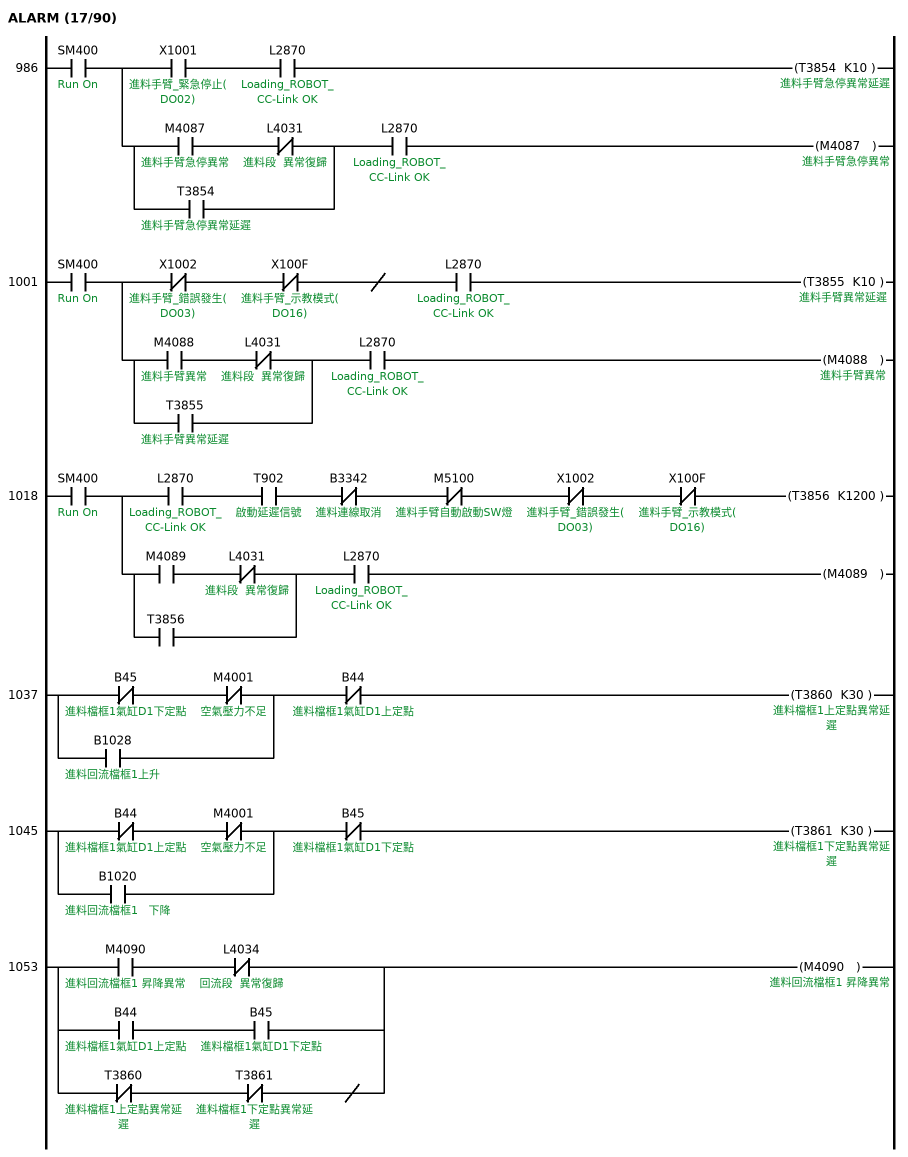
[picture p192: ladder of ALARM, rungs at steps 986 to 1053]
986   LD      SM400  ; Run On
      MPS
      AND     X1001  ; 進料手臂_緊急停止(DO02)
      AND     L2870  ; Loading_ROBOT_  CC-Link OK
      OUT     T3854 K10  ; 進料手臂急停異常延遲
      MPP
      LD      M4087  ; 進料手臂急停異常
      ANI     L4031  ; 進料段  異常復歸
      OR      T3854  ; 進料手臂急停異常延遲
      ANB
      AND     L2870  ; Loading_ROBOT_  CC-Link OK
      OUT     M4087  ; 進料手臂急停異常
1001  LD      SM400  ; Run On
      MPS
      ANI     X1002  ; 進料手臂_錯誤發生(DO03)
      ANI     X100F  ; 進料手臂_示教模式(DO16)
      INV
      AND     L2870  ; Loading_ROBOT_  CC-Link OK
      OUT     T3855 K10  ; 進料手臂異常延遲
      MPP
      LD      M4088  ; 進料手臂異常
      ANI     L4031  ; 進料段  異常復歸
      OR      T3855  ; 進料手臂異常延遲
      ANB
      AND     L2870  ; Loading_ROBOT_  CC-Link OK
      OUT     M4088  ; 進料手臂異常
1018  LD      SM400  ; Run On
      MPS
      AND     L2870  ; Loading_ROBOT_  CC-Link OK
      AND     T902  ; 啟動延遲信號
      ANI     B3342  ; 進料連線取消
      ANI     M5100  ; 進料手臂自動啟動SW燈
      ANI     X1002  ; 進料手臂_錯誤發生(DO03)
      ANI     X100F  ; 進料手臂_示教模式(DO16)
      OUT     T3856 K1200
      MPP
      LD      M4089
      ANI     L4031  ; 進料段  異常復歸
      OR      T3856
      ANB
      AND     L2870  ; Loading_ROBOT_  CC-Link OK
      OUT     M4089
1037  LDI     B45  ; 進料檔框1氣缸D1下定點
      ANI     M4001  ; 空氣壓力不足
      OR      B1028  ; 進料回流檔框1上升
      ANI     B44  ; 進料檔框1氣缸D1上定點
      OUT     T3860 K30  ; 進料檔框1上定點異常延遲
1045  LDI     B44  ; 進料檔框1氣缸D1上定點
      ANI     M4001  ; 空氣壓力不足
      OR      B1020  ; 進料回流檔框1   下降
      ANI     B45  ; 進料檔框1氣缸D1下定點
      OUT     T3861 K30  ; 進料檔框1下定點異常延遲
1053  LD      M4090  ; 進料回流檔框1 昇降異常
      ANI     L4034  ; 回流段  異常復歸
      LD      B44  ; 進料檔框1氣缸D1上定點
      AND     B45  ; 進料檔框1氣缸D1下定點
      ORB
      LDI     T3860  ; 進料檔框1上定點異常延遲
      ANI     T3861  ; 進料檔框1下定點異常延遲
      INV
      ORB
      OUT     M4090  ; 進料回流檔框1 昇降異常
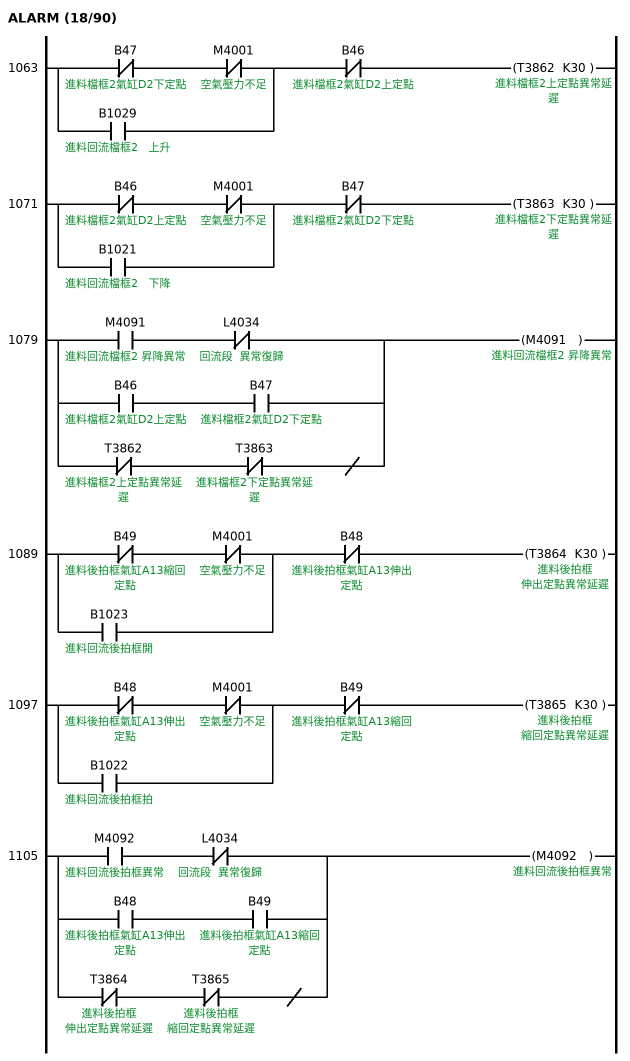
1063  LDI     B47  ; 進料檔框2氣缸D2下定點
      ANI     M4001  ; 空氣壓力不足
      OR      B1029  ; 進料回流檔框2   上升
      ANI     B46  ; 進料檔框2氣缸D2上定點
      OUT     T3862 K30  ; 進料檔框2上定點異常延遲
1071  LDI     B46  ; 進料檔框2氣缸D2上定點
      ANI     M4001  ; 空氣壓力不足
      OR      B1021  ; 進料回流檔框2   下降
      ANI     B47  ; 進料檔框2氣缸D2下定點
      OUT     T3863 K30  ; 進料檔框2下定點異常延遲
1079  LD      M4091  ; 進料回流檔框2 昇降異常
      ANI     L4034  ; 回流段  異常復歸
      LD      B46  ; 進料檔框2氣缸D2上定點
      AND     B47  ; 進料檔框2氣缸D2下定點
      ORB
      LDI     T3862  ; 進料檔框2上定點異常延遲
      ANI     T3863  ; 進料檔框2下定點異常延遲
      INV
      ORB
      OUT     M4091  ; 進料回流檔框2 昇降異常
1089  LDI     B49  ; 進料後拍框氣缸A13縮回定點
      ANI     M4001  ; 空氣壓力不足
      OR      B1023  ; 進料回流後拍框開
      ANI     B48  ; 進料後拍框氣缸A13伸出定點
      OUT     T3864 K30  ; 進料後拍框    伸出定點異常延遲
1097  LDI     B48  ; 進料後拍框氣缸A13伸出定點
      ANI     M4001  ; 空氣壓力不足
      OR      B1022  ; 進料回流後拍框拍
      ANI     B49  ; 進料後拍框氣缸A13縮回定點
      OUT     T3865 K30  ; 進料後拍框    縮回定點異常延遲
1105  LD      M4092  ; 進料回流後拍框異常
      ANI     L4034  ; 回流段  異常復歸
      LD      B48  ; 進料後拍框氣缸A13伸出定點
      AND     B49  ; 進料後拍框氣缸A13縮回定點
      ORB
      LDI     T3864  ; 進料後拍框    伸出定點異常延遲
      ANI     T3865  ; 進料後拍框    縮回定點異常延遲
      INV
      ORB
      OUT     M4092  ; 進料回流後拍框異常
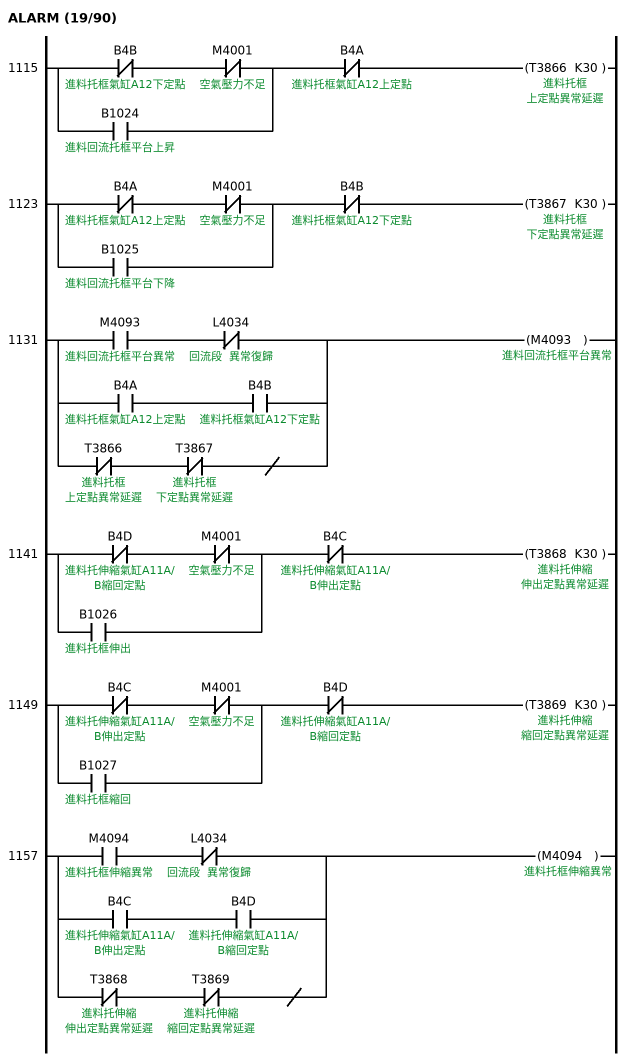
1115  LDI     B4B  ; 進料托框氣缸A12下定點
      ANI     M4001  ; 空氣壓力不足
      OR      B1024  ; 進料回流托框平台上昇
      ANI     B4A  ; 進料托框氣缸A12上定點
      OUT     T3866 K30  ; 進料托框    上定點異常延遲
1123  LDI     B4A  ; 進料托框氣缸A12上定點
      ANI     M4001  ; 空氣壓力不足
      OR      B1025  ; 進料回流托框平台下降
      ANI     B4B  ; 進料托框氣缸A12下定點
      OUT     T3867 K30  ; 進料托框    下定點異常延遲
1131  LD      M4093  ; 進料回流托框平台異常
      ANI     L4034  ; 回流段  異常復歸
      LD      B4A  ; 進料托框氣缸A12上定點
      AND     B4B  ; 進料托框氣缸A12下定點
      ORB
      LDI     T3866  ; 進料托框    上定點異常延遲
      ANI     T3867  ; 進料托框    下定點異常延遲
      INV
      ORB
      OUT     M4093  ; 進料回流托框平台異常
1141  LDI     B4D  ; 進料托伸縮氣缸A11A/B縮回定點
      ANI     M4001  ; 空氣壓力不足
      OR      B1026  ; 進料托框伸出
      ANI     B4C  ; 進料托伸縮氣缸A11A/B伸出定點
      OUT     T3868 K30  ; 進料托伸縮    伸出定點異常延遲
1149  LDI     B4C  ; 進料托伸縮氣缸A11A/B伸出定點
      ANI     M4001  ; 空氣壓力不足
      OR      B1027  ; 進料托框縮回
      ANI     B4D  ; 進料托伸縮氣缸A11A/B縮回定點
      OUT     T3869 K30  ; 進料托伸縮    縮回定點異常延遲
1157  LD      M4094  ; 進料托框伸縮異常
      ANI     L4034  ; 回流段  異常復歸
      LD      B4C  ; 進料托伸縮氣缸A11A/B伸出定點
      AND     B4D  ; 進料托伸縮氣缸A11A/B縮回定點
      ORB
      LDI     T3868  ; 進料托伸縮    伸出定點異常延遲
      ANI     T3869  ; 進料托伸縮    縮回定點異常延遲
      INV
      ORB
      OUT     M4094  ; 進料托框伸縮異常
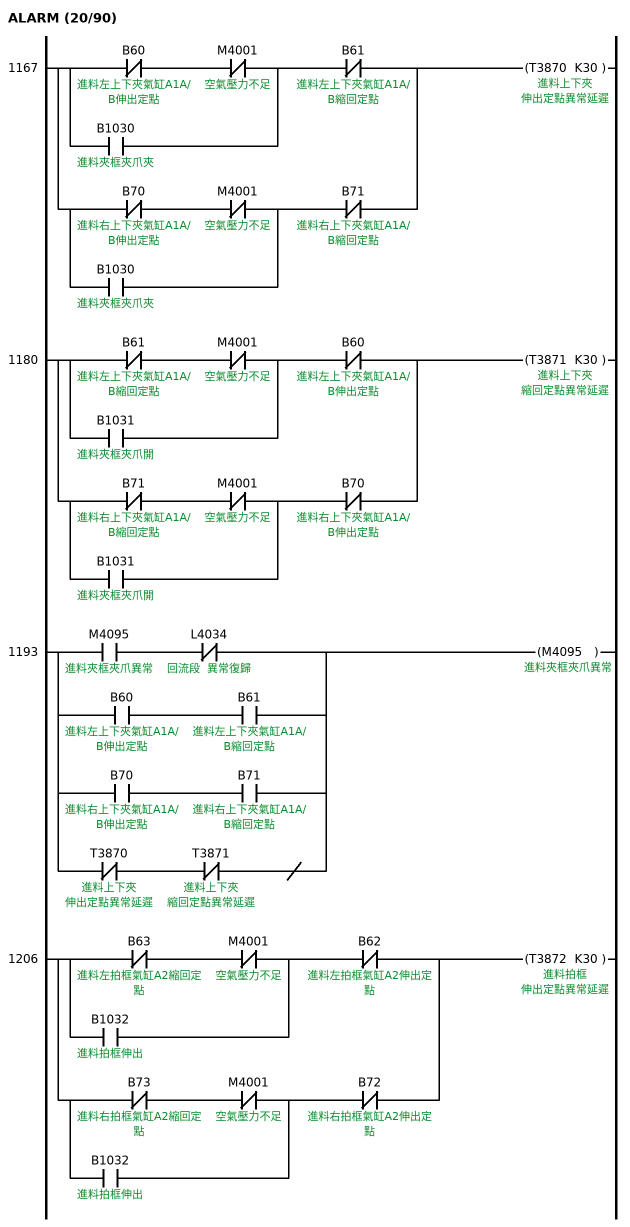
1167  LDI     B60  ; 進料左上下夾氣缸A1A/B伸出定點
      ANI     M4001  ; 空氣壓力不足
      OR      B1030  ; 進料夾框夾爪夾
      ANI     B61  ; 進料左上下夾氣缸A1A/B縮回定點
      LDI     B70  ; 進料右上下夾氣缸A1A/B伸出定點
      ANI     M4001  ; 空氣壓力不足
      OR      B1030  ; 進料夾框夾爪夾
      ANI     B71  ; 進料右上下夾氣缸A1A/B縮回定點
      ORB
      OUT     T3870 K30  ; 進料上下夾    伸出定點異常延遲
1180  LDI     B61  ; 進料左上下夾氣缸A1A/B縮回定點
      ANI     M4001  ; 空氣壓力不足
      OR      B1031  ; 進料夾框夾爪開
      ANI     B60  ; 進料左上下夾氣缸A1A/B伸出定點
      LDI     B71  ; 進料右上下夾氣缸A1A/B縮回定點
      ANI     M4001  ; 空氣壓力不足
      OR      B1031  ; 進料夾框夾爪開
      ANI     B70  ; 進料右上下夾氣缸A1A/B伸出定點
      ORB
      OUT     T3871 K30  ; 進料上下夾    縮回定點異常延遲
1193  LD      M4095  ; 進料夾框夾爪異常
      ANI     L4034  ; 回流段  異常復歸
      LD      B60  ; 進料左上下夾氣缸A1A/B伸出定點
      AND     B61  ; 進料左上下夾氣缸A1A/B縮回定點
      ORB
      LD      B70  ; 進料右上下夾氣缸A1A/B伸出定點
      AND     B71  ; 進料右上下夾氣缸A1A/B縮回定點
      ORB
      LDI     T3870  ; 進料上下夾    伸出定點異常延遲
      ANI     T3871  ; 進料上下夾    縮回定點異常延遲
      INV
      ORB
      OUT     M4095  ; 進料夾框夾爪異常
1206  LDI     B63  ; 進料左拍框氣缸A2縮回定點
      ANI     M4001  ; 空氣壓力不足
      OR      B1032  ; 進料拍框伸出
      ANI     B62  ; 進料左拍框氣缸A2伸出定點
      LDI     B73  ; 進料右拍框氣缸A2縮回定點
      ANI     M4001  ; 空氣壓力不足
      OR      B1032  ; 進料拍框伸出
      ANI     B72  ; 進料右拍框氣缸A2伸出定點
      ORB
      OUT     T3872 K30  ; 進料拍框    伸出定點異常延遲
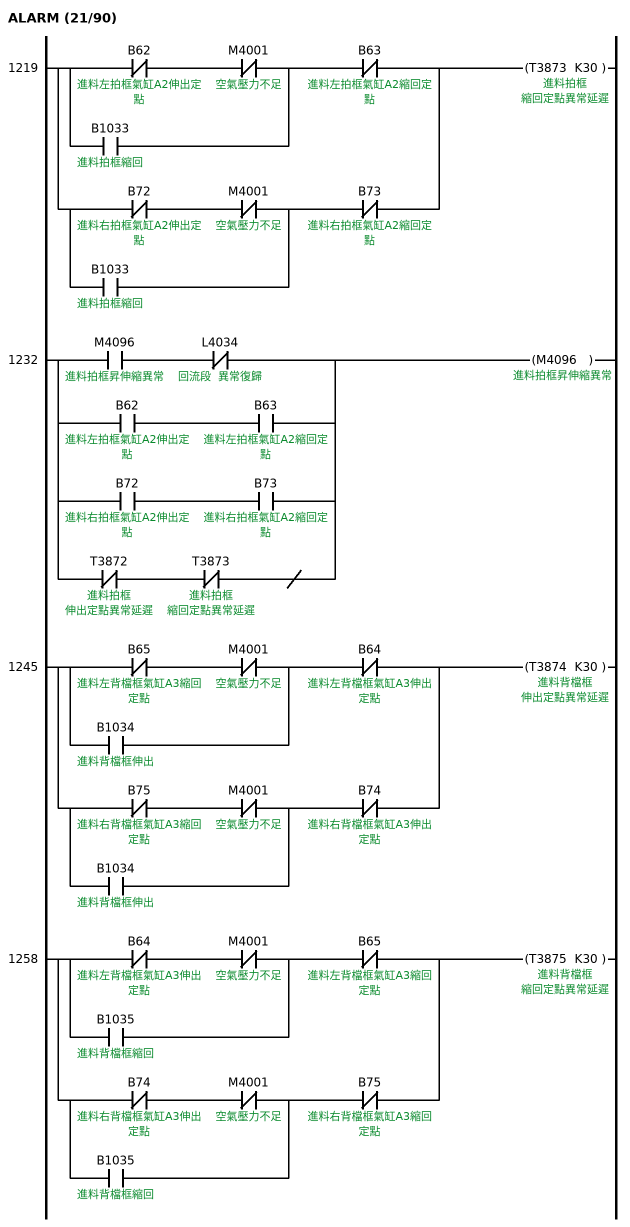
1219  LDI     B62  ; 進料左拍框氣缸A2伸出定點
      ANI     M4001  ; 空氣壓力不足
      OR      B1033  ; 進料拍框縮回
      ANI     B63  ; 進料左拍框氣缸A2縮回定點
      LDI     B72  ; 進料右拍框氣缸A2伸出定點
      ANI     M4001  ; 空氣壓力不足
      OR      B1033  ; 進料拍框縮回
      ANI     B73  ; 進料右拍框氣缸A2縮回定點
      ORB
      OUT     T3873 K30  ; 進料拍框    縮回定點異常延遲
1232  LD      M4096  ; 進料拍框昇伸縮異常
      ANI     L4034  ; 回流段  異常復歸
      LD      B62  ; 進料左拍框氣缸A2伸出定點
      AND     B63  ; 進料左拍框氣缸A2縮回定點
      ORB
      LD      B72  ; 進料右拍框氣缸A2伸出定點
      AND     B73  ; 進料右拍框氣缸A2縮回定點
      ORB
      LDI     T3872  ; 進料拍框    伸出定點異常延遲
      ANI     T3873  ; 進料拍框    縮回定點異常延遲
      INV
      ORB
      OUT     M4096  ; 進料拍框昇伸縮異常
1245  LDI     B65  ; 進料左背檔框氣缸A3縮回定點
      ANI     M4001  ; 空氣壓力不足
      OR      B1034  ; 進料背檔框伸出
      ANI     B64  ; 進料左背檔框氣缸A3伸出定點
      LDI     B75  ; 進料右背檔框氣缸A3縮回定點
      ANI     M4001  ; 空氣壓力不足
      OR      B1034  ; 進料背檔框伸出
      ANI     B74  ; 進料右背檔框氣缸A3伸出定點
      ORB
      OUT     T3874 K30  ; 進料背檔框    伸出定點異常延遲
1258  LDI     B64  ; 進料左背檔框氣缸A3伸出定點
      ANI     M4001  ; 空氣壓力不足
      OR      B1035  ; 進料背檔框縮回
      ANI     B65  ; 進料左背檔框氣缸A3縮回定點
      LDI     B74  ; 進料右背檔框氣缸A3伸出定點
      ANI     M4001  ; 空氣壓力不足
      OR      B1035  ; 進料背檔框縮回
      ANI     B75  ; 進料右背檔框氣缸A3縮回定點
      ORB
      OUT     T3875 K30  ; 進料背檔框    縮回定點異常延遲
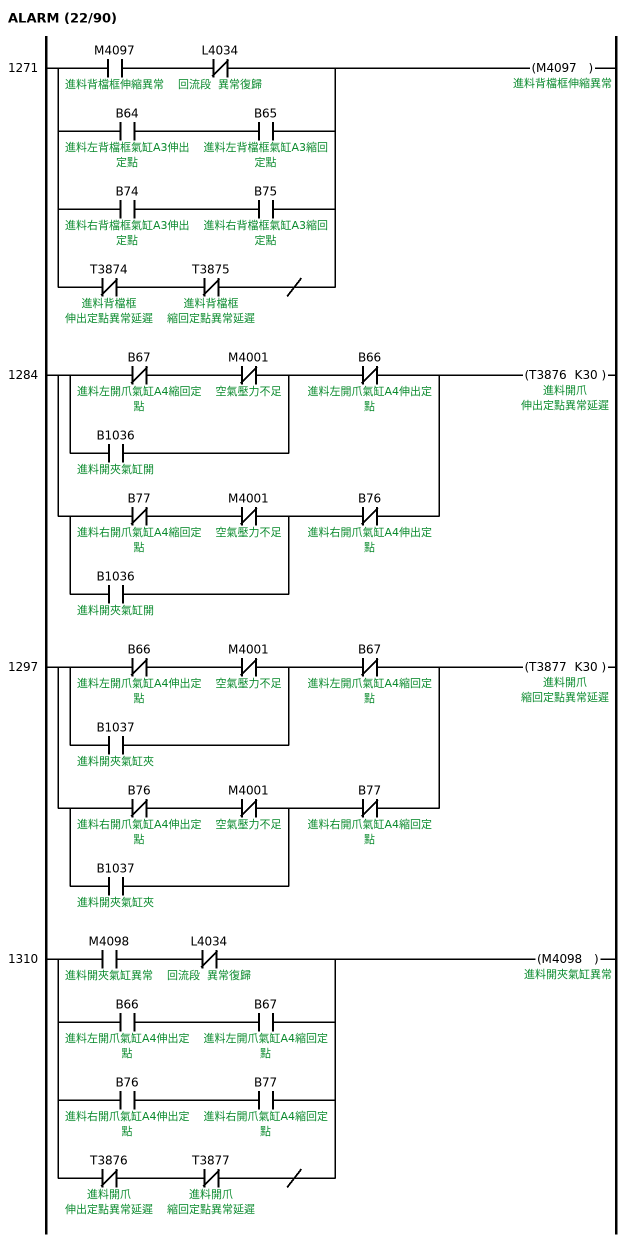
1271  LD      M4097  ; 進料背檔框伸縮異常
      ANI     L4034  ; 回流段  異常復歸
      LD      B64  ; 進料左背檔框氣缸A3伸出定點
      AND     B65  ; 進料左背檔框氣缸A3縮回定點
      ORB
      LD      B74  ; 進料右背檔框氣缸A3伸出定點
      AND     B75  ; 進料右背檔框氣缸A3縮回定點
      ORB
      LDI     T3874  ; 進料背檔框    伸出定點異常延遲
      ANI     T3875  ; 進料背檔框    縮回定點異常延遲
      INV
      ORB
      OUT     M4097  ; 進料背檔框伸縮異常
1284  LDI     B67  ; 進料左開爪氣缸A4縮回定點
      ANI     M4001  ; 空氣壓力不足
      OR      B1036  ; 進料開夾氣缸開
      ANI     B66  ; 進料左開爪氣缸A4伸出定點
      LDI     B77  ; 進料右開爪氣缸A4縮回定點
      ANI     M4001  ; 空氣壓力不足
      OR      B1036  ; 進料開夾氣缸開
      ANI     B76  ; 進料右開爪氣缸A4伸出定點
      ORB
      OUT     T3876 K30  ; 進料開爪    伸出定點異常延遲
1297  LDI     B66  ; 進料左開爪氣缸A4伸出定點
      ANI     M4001  ; 空氣壓力不足
      OR      B1037  ; 進料開夾氣缸夾
      ANI     B67  ; 進料左開爪氣缸A4縮回定點
      LDI     B76  ; 進料右開爪氣缸A4伸出定點
      ANI     M4001  ; 空氣壓力不足
      OR      B1037  ; 進料開夾氣缸夾
      ANI     B77  ; 進料右開爪氣缸A4縮回定點
      ORB
      OUT     T3877 K30  ; 進料開爪    縮回定點異常延遲
1310  LD      M4098  ; 進料開夾氣缸異常
      ANI     L4034  ; 回流段  異常復歸
      LD      B66  ; 進料左開爪氣缸A4伸出定點
      AND     B67  ; 進料左開爪氣缸A4縮回定點
      ORB
      LD      B76  ; 進料右開爪氣缸A4伸出定點
      AND     B77  ; 進料右開爪氣缸A4縮回定點
      ORB
      LDI     T3876  ; 進料開爪    伸出定點異常延遲
      ANI     T3877  ; 進料開爪    縮回定點異常延遲
      INV
      ORB
      OUT     M4098  ; 進料開夾氣缸異常
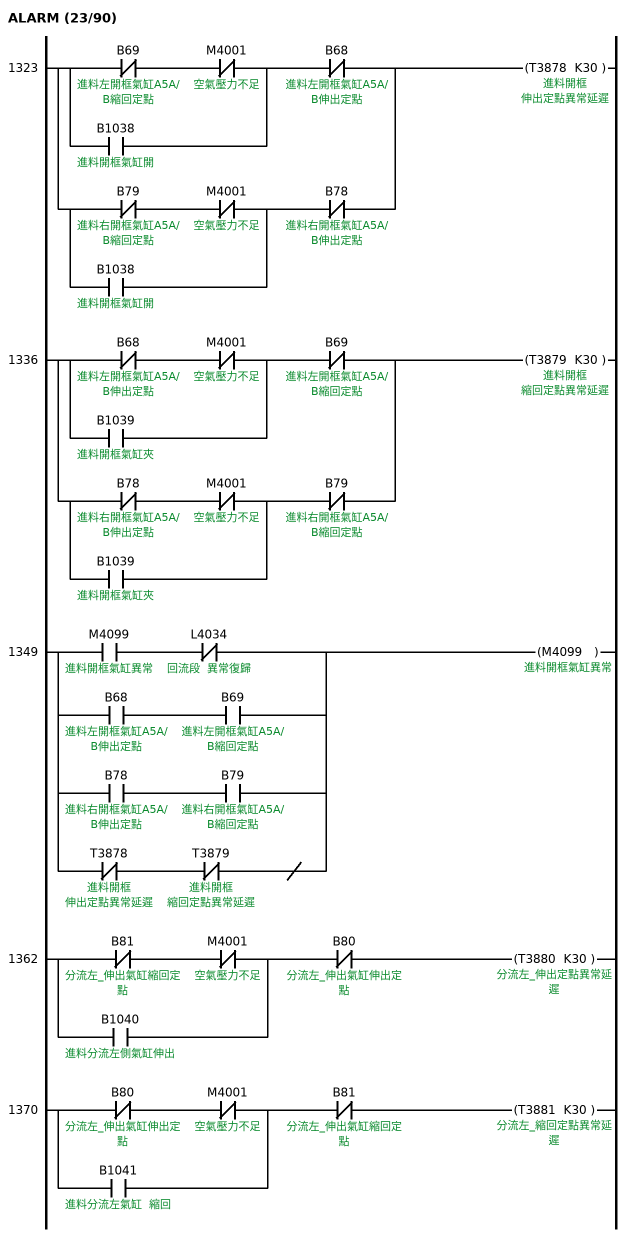
1323  LDI     B69  ; 進料左開框氣缸A5A/B縮回定點
      ANI     M4001  ; 空氣壓力不足
      OR      B1038  ; 進料開框氣缸開
      ANI     B68  ; 進料左開框氣缸A5A/B伸出定點
      LDI     B79  ; 進料右開框氣缸A5A/B縮回定點
      ANI     M4001  ; 空氣壓力不足
      OR      B1038  ; 進料開框氣缸開
      ANI     B78  ; 進料右開框氣缸A5A/B伸出定點
      ORB
      OUT     T3878 K30  ; 進料開框    伸出定點異常延遲
1336  LDI     B68  ; 進料左開框氣缸A5A/B伸出定點
      ANI     M4001  ; 空氣壓力不足
      OR      B1039  ; 進料開框氣缸夾
      ANI     B69  ; 進料左開框氣缸A5A/B縮回定點
      LDI     B78  ; 進料右開框氣缸A5A/B伸出定點
      ANI     M4001  ; 空氣壓力不足
      OR      B1039  ; 進料開框氣缸夾
      ANI     B79  ; 進料右開框氣缸A5A/B縮回定點
      ORB
      OUT     T3879 K30  ; 進料開框    縮回定點異常延遲
1349  LD      M4099  ; 進料開框氣缸異常
      ANI     L4034  ; 回流段  異常復歸
      LD      B68  ; 進料左開框氣缸A5A/B伸出定點
      AND     B69  ; 進料左開框氣缸A5A/B縮回定點
      ORB
      LD      B78  ; 進料右開框氣缸A5A/B伸出定點
      AND     B79  ; 進料右開框氣缸A5A/B縮回定點
      ORB
      LDI     T3878  ; 進料開框    伸出定點異常延遲
      ANI     T3879  ; 進料開框    縮回定點異常延遲
      INV
      ORB
      OUT     M4099  ; 進料開框氣缸異常
1362  LDI     B81  ; 分流左_伸出氣缸縮回定點
      ANI     M4001  ; 空氣壓力不足
      OR      B1040  ; 進料分流左側氣缸伸出
      ANI     B80  ; 分流左_伸出氣缸伸出定點
      OUT     T3880 K30  ; 分流左_伸出定點異常延遲
1370  LDI     B80  ; 分流左_伸出氣缸伸出定點
      ANI     M4001  ; 空氣壓力不足
      OR      B1041  ; 進料分流左氣缸  縮回
      ANI     B81  ; 分流左_伸出氣缸縮回定點
      OUT     T3881 K30  ; 分流左_縮回定點異常延遲
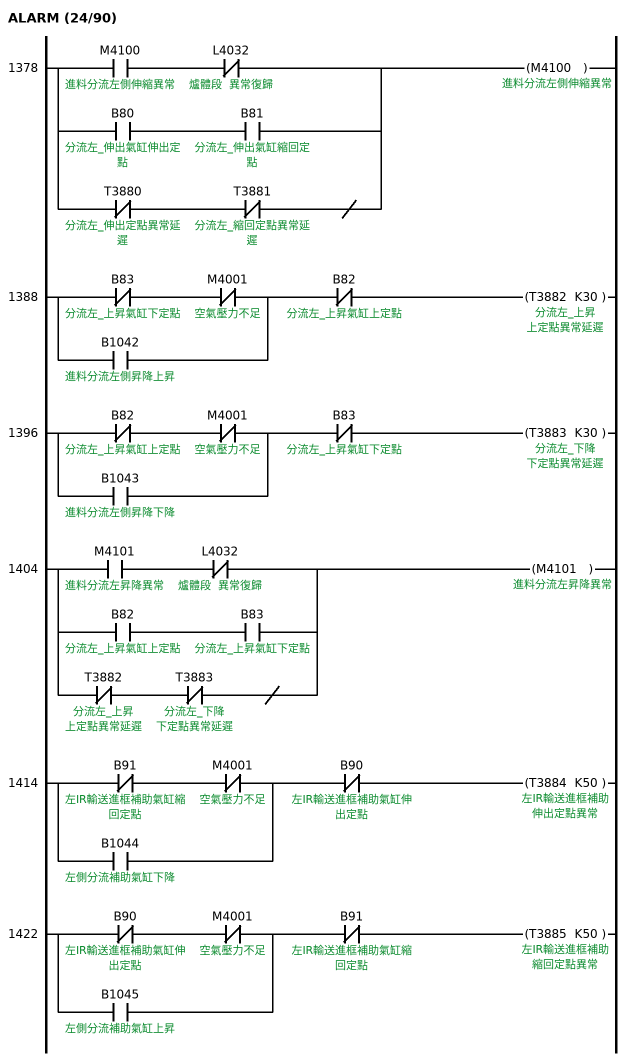
1378  LD      M4100  ; 進料分流左側伸縮異常
      ANI     L4032  ; 爐體段  異常復歸
      LD      B80  ; 分流左_伸出氣缸伸出定點
      AND     B81  ; 分流左_伸出氣缸縮回定點
      ORB
      LDI     T3880  ; 分流左_伸出定點異常延遲
      ANI     T3881  ; 分流左_縮回定點異常延遲
      INV
      ORB
      OUT     M4100  ; 進料分流左側伸縮異常
1388  LDI     B83  ; 分流左_上昇氣缸下定點
      ANI     M4001  ; 空氣壓力不足
      OR      B1042  ; 進料分流左側昇降上昇
      ANI     B82  ; 分流左_上昇氣缸上定點
      OUT     T3882 K30  ; 分流左_上昇    上定點異常延遲
1396  LDI     B82  ; 分流左_上昇氣缸上定點
      ANI     M4001  ; 空氣壓力不足
      OR      B1043  ; 進料分流左側昇降下降
      ANI     B83  ; 分流左_上昇氣缸下定點
      OUT     T3883 K30  ; 分流左_下降    下定點異常延遲
1404  LD      M4101  ; 進料分流左昇降異常
      ANI     L4032  ; 爐體段  異常復歸
      LD      B82  ; 分流左_上昇氣缸上定點
      AND     B83  ; 分流左_上昇氣缸下定點
      ORB
      LDI     T3882  ; 分流左_上昇    上定點異常延遲
      ANI     T3883  ; 分流左_下降    下定點異常延遲
      INV
      ORB
      OUT     M4101  ; 進料分流左昇降異常
1414  LDI     B91  ; 左IR輸送進框補助氣缸縮回定點
      ANI     M4001  ; 空氣壓力不足
      OR      B1044  ; 左側分流補助氣缸下降
      ANI     B90  ; 左IR輸送進框補助氣缸伸出定點
      OUT     T3884 K50  ; 左IR輸送進框補助    伸出定點異常
1422  LDI     B90  ; 左IR輸送進框補助氣缸伸出定點
      ANI     M4001  ; 空氣壓力不足
      OR      B1045  ; 左側分流補助氣缸上昇
      ANI     B91  ; 左IR輸送進框補助氣缸縮回定點
      OUT     T3885 K50  ; 左IR輸送進框補助    縮回定點異常
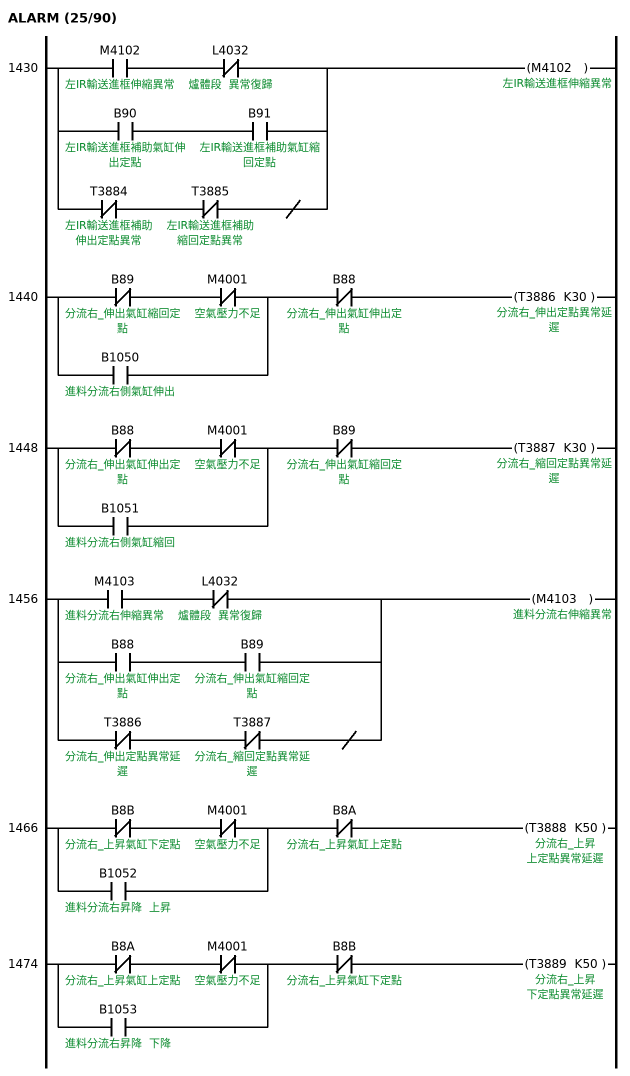
1430  LD      M4102  ; 左IR輸送進框伸縮異常
      ANI     L4032  ; 爐體段  異常復歸
      LD      B90  ; 左IR輸送進框補助氣缸伸出定點
      AND     B91  ; 左IR輸送進框補助氣缸縮回定點
      ORB
      LDI     T3884  ; 左IR輸送進框補助    伸出定點異常
      ANI     T3885  ; 左IR輸送進框補助    縮回定點異常
      INV
      ORB
      OUT     M4102  ; 左IR輸送進框伸縮異常
1440  LDI     B89  ; 分流右_伸出氣缸縮回定點
      ANI     M4001  ; 空氣壓力不足
      OR      B1050  ; 進料分流右側氣缸伸出
      ANI     B88  ; 分流右_伸出氣缸伸出定點
      OUT     T3886 K30  ; 分流右_伸出定點異常延遲
1448  LDI     B88  ; 分流右_伸出氣缸伸出定點
      ANI     M4001  ; 空氣壓力不足
      OR      B1051  ; 進料分流右側氣缸縮回
      ANI     B89  ; 分流右_伸出氣缸縮回定點
      OUT     T3887 K30  ; 分流右_縮回定點異常延遲
1456  LD      M4103  ; 進料分流右伸縮異常
      ANI     L4032  ; 爐體段  異常復歸
      LD      B88  ; 分流右_伸出氣缸伸出定點
      AND     B89  ; 分流右_伸出氣缸縮回定點
      ORB
      LDI     T3886  ; 分流右_伸出定點異常延遲
      ANI     T3887  ; 分流右_縮回定點異常延遲
      INV
      ORB
      OUT     M4103  ; 進料分流右伸縮異常
1466  LDI     B8B  ; 分流右_上昇氣缸下定點
      ANI     M4001  ; 空氣壓力不足
      OR      B1052  ; 進料分流右昇降  上昇
      ANI     B8A  ; 分流右_上昇氣缸上定點
      OUT     T3888 K50  ; 分流右_上昇    上定點異常延遲
1474  LDI     B8A  ; 分流右_上昇氣缸上定點
      ANI     M4001  ; 空氣壓力不足
      OR      B1053  ; 進料分流右昇降  下降
      ANI     B8B  ; 分流右_上昇氣缸下定點
      OUT     T3889 K50  ; 分流右_上昇    下定點異常延遲
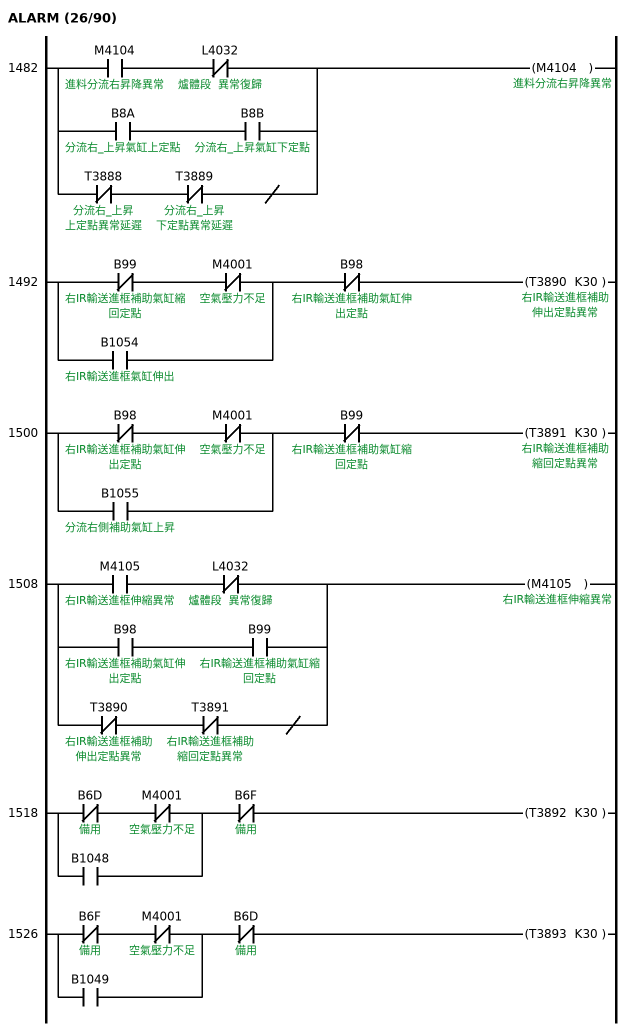
1482  LD      M4104  ; 進料分流右昇降異常
      ANI     L4032  ; 爐體段  異常復歸
      LD      B8A  ; 分流右_上昇氣缸上定點
      AND     B8B  ; 分流右_上昇氣缸下定點
      ORB
      LDI     T3888  ; 分流右_上昇    上定點異常延遲
      ANI     T3889  ; 分流右_上昇    下定點異常延遲
      INV
      ORB
      OUT     M4104  ; 進料分流右昇降異常
1492  LDI     B99  ; 右IR輸送進框補助氣缸縮回定點
      ANI     M4001  ; 空氣壓力不足
      OR      B1054  ; 右IR輸送進框氣缸伸出
      ANI     B98  ; 右IR輸送進框補助氣缸伸出定點
      OUT     T3890 K30  ; 右IR輸送進框補助    伸出定點異常
1500  LDI     B98  ; 右IR輸送進框補助氣缸伸出定點
      ANI     M4001  ; 空氣壓力不足
      OR      B1055  ; 分流右側補助氣缸上昇
      ANI     B99  ; 右IR輸送進框補助氣缸縮回定點
      OUT     T3891 K30  ; 右IR輸送進框補助    縮回定點異常
1508  LD      M4105  ; 右IR輸送進框伸縮異常
      ANI     L4032  ; 爐體段  異常復歸
      LD      B98  ; 右IR輸送進框補助氣缸伸出定點
      AND     B99  ; 右IR輸送進框補助氣缸縮回定點
      ORB
      LDI     T3890  ; 右IR輸送進框補助    伸出定點異常
      ANI     T3891  ; 右IR輸送進框補助    縮回定點異常
      INV
      ORB
      OUT     M4105  ; 右IR輸送進框伸縮異常
1518  LDI     B6D  ; 備用
      ANI     M4001  ; 空氣壓力不足
      OR      B1048
      ANI     B6F  ; 備用
      OUT     T3892 K30
1526  LDI     B6F  ; 備用
      ANI     M4001  ; 空氣壓力不足
      OR      B1049
      ANI     B6D  ; 備用
      OUT     T3893 K30
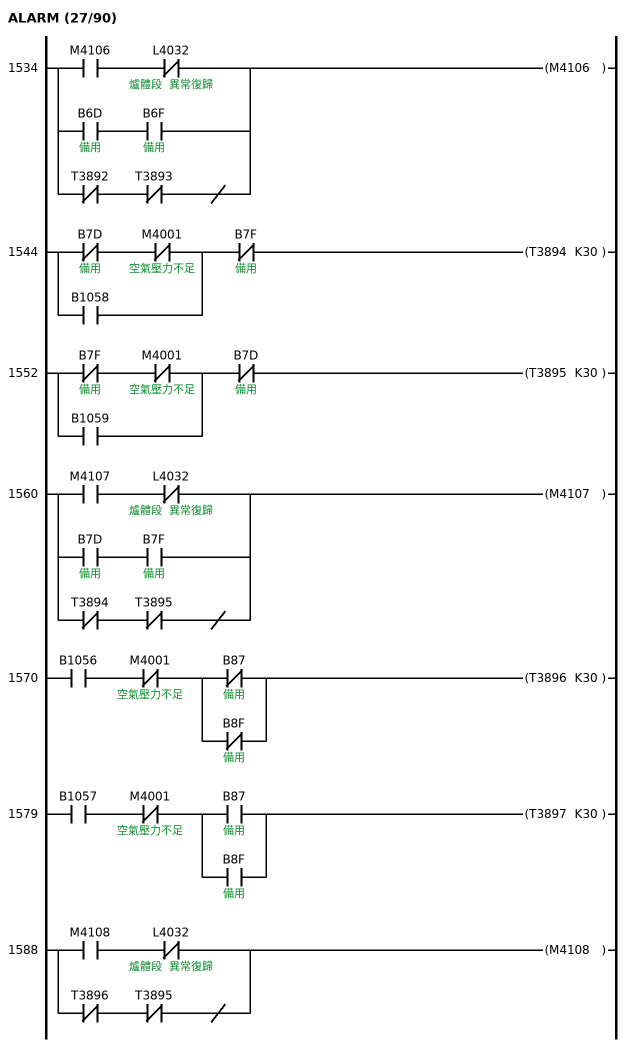
1534  LD      M4106
      ANI     L4032  ; 爐體段  異常復歸
      LD      B6D  ; 備用
      AND     B6F  ; 備用
      ORB
      LDI     T3892
      ANI     T3893
      INV
      ORB
      OUT     M4106
1544  LDI     B7D  ; 備用
      ANI     M4001  ; 空氣壓力不足
      OR      B1058
      ANI     B7F  ; 備用
      OUT     T3894 K30
1552  LDI     B7F  ; 備用
      ANI     M4001  ; 空氣壓力不足
      OR      B1059
      ANI     B7D  ; 備用
      OUT     T3895 K30
1560  LD      M4107
      ANI     L4032  ; 爐體段  異常復歸
      LD      B7D  ; 備用
      AND     B7F  ; 備用
      ORB
      LDI     T3894
      ANI     T3895
      INV
      ORB
      OUT     M4107
1570  LD      B1056
      ANI     M4001  ; 空氣壓力不足
      LDI     B87  ; 備用
      ORI     B8F  ; 備用
      ANB
      OUT     T3896 K30
1579  LD      B1057
      ANI     M4001  ; 空氣壓力不足
      LD      B87  ; 備用
      OR      B8F  ; 備用
      ANB
      OUT     T3897 K30
1588  LD      M4108
      ANI     L4032  ; 爐體段  異常復歸
      LDI     T3896
      ANI     T3895
      INV
      ORB
      OUT     M4108
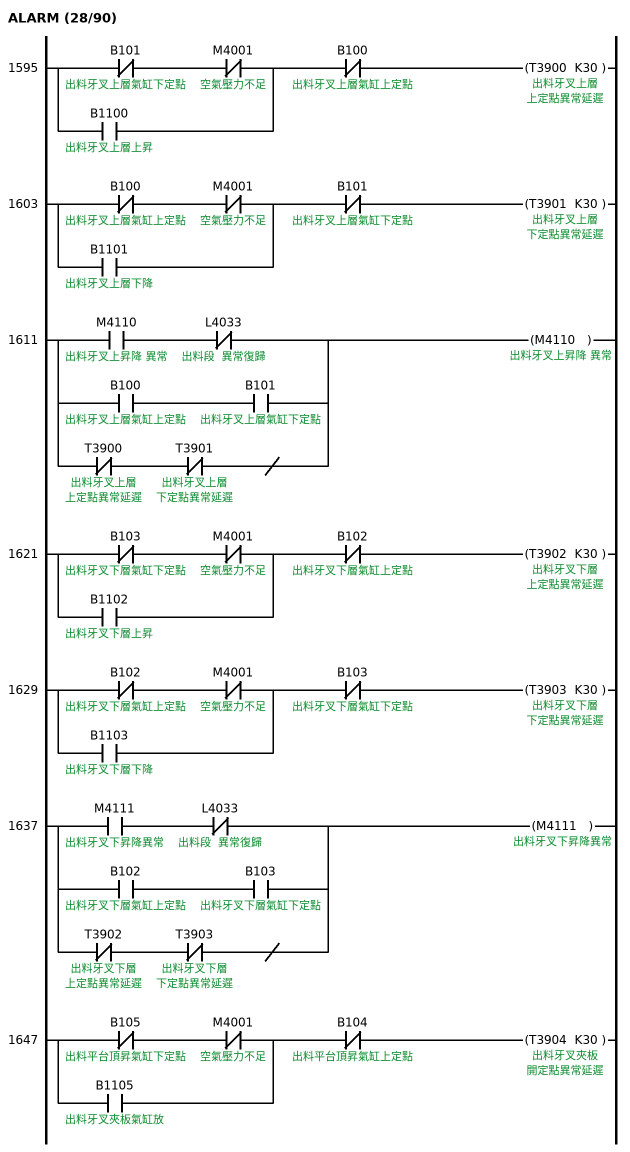
1595  LDI     B101  ; 出料牙叉上層氣缸下定點
      ANI     M4001  ; 空氣壓力不足
      OR      B1100  ; 出料牙叉上層上昇
      ANI     B100  ; 出料牙叉上層氣缸上定點
      OUT     T3900 K30  ; 出料牙叉上層    上定點異常延遲
1603  LDI     B100  ; 出料牙叉上層氣缸上定點
      ANI     M4001  ; 空氣壓力不足
      OR      B1101  ; 出料牙叉上層下降
      ANI     B101  ; 出料牙叉上層氣缸下定點
      OUT     T3901 K30  ; 出料牙叉上層    下定點異常延遲
1611  LD      M4110  ; 出料牙叉上昇降 異常
      ANI     L4033  ; 出料段  異常復歸
      LD      B100  ; 出料牙叉上層氣缸上定點
      AND     B101  ; 出料牙叉上層氣缸下定點
      ORB
      LDI     T3900  ; 出料牙叉上層    上定點異常延遲
      ANI     T3901  ; 出料牙叉上層    下定點異常延遲
      INV
      ORB
      OUT     M4110  ; 出料牙叉上昇降 異常
1621  LDI     B103  ; 出料牙叉下層氣缸下定點
      ANI     M4001  ; 空氣壓力不足
      OR      B1102  ; 出料牙叉下層上昇
      ANI     B102  ; 出料牙叉下層氣缸上定點
      OUT     T3902 K30  ; 出料牙叉下層    上定點異常延遲
1629  LDI     B102  ; 出料牙叉下層氣缸上定點
      ANI     M4001  ; 空氣壓力不足
      OR      B1103  ; 出料牙叉下層下降
      ANI     B103  ; 出料牙叉下層氣缸下定點
      OUT     T3903 K30  ; 出料牙叉下層    下定點異常延遲
1637  LD      M4111  ; 出料牙叉下昇降異常
      ANI     L4033  ; 出料段  異常復歸
      LD      B102  ; 出料牙叉下層氣缸上定點
      AND     B103  ; 出料牙叉下層氣缸下定點
      ORB
      LDI     T3902  ; 出料牙叉下層    上定點異常延遲
      ANI     T3903  ; 出料牙叉下層    下定點異常延遲
      INV
      ORB
      OUT     M4111  ; 出料牙叉下昇降異常
1647  LDI     B105  ; 出料平台頂昇氣缸下定點
      ANI     M4001  ; 空氣壓力不足
      OR      B1105  ; 出料牙叉夾板氣缸放
      ANI     B104  ; 出料平台頂昇氣缸上定點
      OUT     T3904 K30  ; 出料牙叉夾板    開定點異常延遲
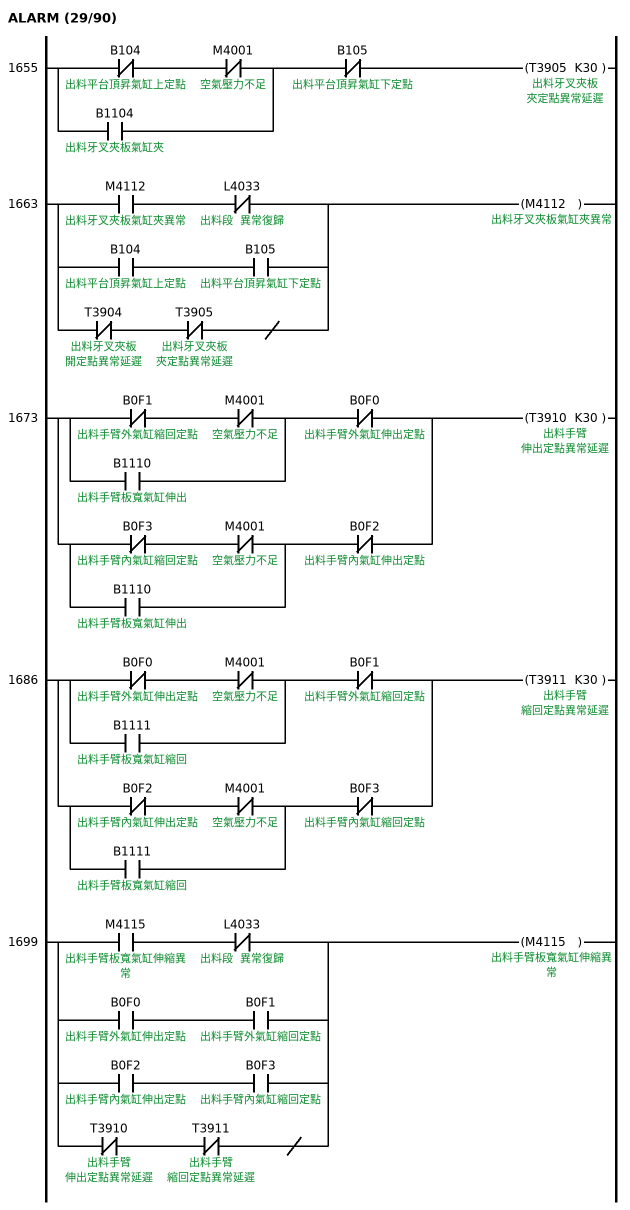
1655  LDI     B104  ; 出料平台頂昇氣缸上定點
      ANI     M4001  ; 空氣壓力不足
      OR      B1104  ; 出料牙叉夾板氣缸夾
      ANI     B105  ; 出料平台頂昇氣缸下定點
      OUT     T3905 K30  ; 出料牙叉夾板    夾定點異常延遲
1663  LD      M4112  ; 出料牙叉夾板氣缸夾異常
      ANI     L4033  ; 出料段  異常復歸
      LD      B104  ; 出料平台頂昇氣缸上定點
      AND     B105  ; 出料平台頂昇氣缸下定點
      ORB
      LDI     T3904  ; 出料牙叉夾板    開定點異常延遲
      ANI     T3905  ; 出料牙叉夾板    夾定點異常延遲
      INV
      ORB
      OUT     M4112  ; 出料牙叉夾板氣缸夾異常
1673  LDI     B0F1  ; 出料手臂外氣缸縮回定點
      ANI     M4001  ; 空氣壓力不足
      OR      B1110  ; 出料手臂板寬氣缸伸出
      ANI     B0F0  ; 出料手臂外氣缸伸出定點
      LDI     B0F3  ; 出料手臂內氣缸縮回定點
      ANI     M4001  ; 空氣壓力不足
      OR      B1110  ; 出料手臂板寬氣缸伸出
      ANI     B0F2  ; 出料手臂內氣缸伸出定點
      ORB
      OUT     T3910 K30  ; 出料手臂    伸出定點異常延遲
1686  LDI     B0F0  ; 出料手臂外氣缸伸出定點
      ANI     M4001  ; 空氣壓力不足
      OR      B1111  ; 出料手臂板寬氣缸縮回
      ANI     B0F1  ; 出料手臂外氣缸縮回定點
      LDI     B0F2  ; 出料手臂內氣缸伸出定點
      ANI     M4001  ; 空氣壓力不足
      OR      B1111  ; 出料手臂板寬氣缸縮回
      ANI     B0F3  ; 出料手臂內氣缸縮回定點
      ORB
      OUT     T3911 K30  ; 出料手臂    縮回定點異常延遲
1699  LD      M4115  ; 出料手臂板寬氣缸伸縮異常
      ANI     L4033  ; 出料段  異常復歸
      LD      B0F0  ; 出料手臂外氣缸伸出定點
      AND     B0F1  ; 出料手臂外氣缸縮回定點
      ORB
      LD      B0F2  ; 出料手臂內氣缸伸出定點
      AND     B0F3  ; 出料手臂內氣缸縮回定點
      ORB
      LDI     T3910  ; 出料手臂    伸出定點異常延遲
      ANI     T3911  ; 出料手臂    縮回定點異常延遲
      INV
      ORB
      OUT     M4115  ; 出料手臂板寬氣缸伸縮異常
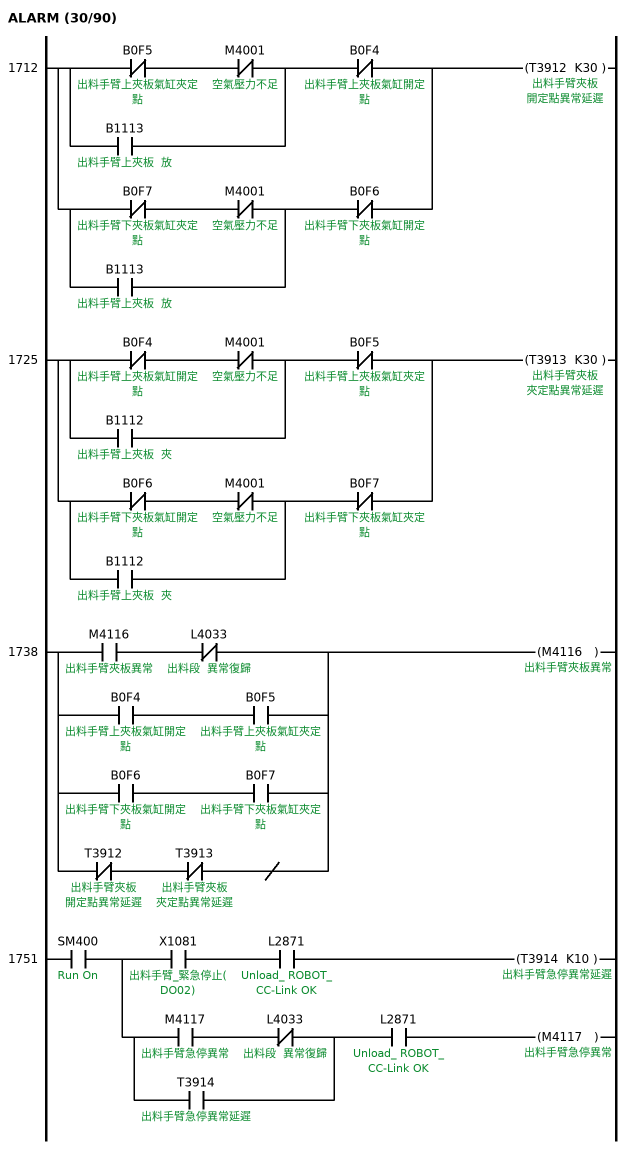
1712  LDI     B0F5  ; 出料手臂上夾板氣缸夾定點
      ANI     M4001  ; 空氣壓力不足
      OR      B1113  ; 出料手臂上夾板  放
      ANI     B0F4  ; 出料手臂上夾板氣缸開定點
      LDI     B0F7  ; 出料手臂下夾板氣缸夾定點
      ANI     M4001  ; 空氣壓力不足
      OR      B1113  ; 出料手臂上夾板  放
      ANI     B0F6  ; 出料手臂下夾板氣缸開定點
      ORB
      OUT     T3912 K30  ; 出料手臂夾板    開定點異常延遲
1725  LDI     B0F4  ; 出料手臂上夾板氣缸開定點
      ANI     M4001  ; 空氣壓力不足
      OR      B1112  ; 出料手臂上夾板  夾
      ANI     B0F5  ; 出料手臂上夾板氣缸夾定點
      LDI     B0F6  ; 出料手臂下夾板氣缸開定點
      ANI     M4001  ; 空氣壓力不足
      OR      B1112  ; 出料手臂上夾板  夾
      ANI     B0F7  ; 出料手臂下夾板氣缸夾定點
      ORB
      OUT     T3913 K30  ; 出料手臂夾板    夾定點異常延遲
1738  LD      M4116  ; 出料手臂夾板異常
      ANI     L4033  ; 出料段  異常復歸
      LD      B0F4  ; 出料手臂上夾板氣缸開定點
      AND     B0F5  ; 出料手臂上夾板氣缸夾定點
      ORB
      LD      B0F6  ; 出料手臂下夾板氣缸開定點
      AND     B0F7  ; 出料手臂下夾板氣缸夾定點
      ORB
      LDI     T3912  ; 出料手臂夾板    開定點異常延遲
      ANI     T3913  ; 出料手臂夾板    夾定點異常延遲
      INV
      ORB
      OUT     M4116  ; 出料手臂夾板異常
1751  LD      SM400  ; Run On
      MPS
      AND     X1081  ; 出料手臂_緊急停止(DO02)
      AND     L2871  ; Unload_ ROBOT_  CC-Link OK
      OUT     T3914 K10  ; 出料手臂急停異常延遲
      MPP
      LD      M4117  ; 出料手臂急停異常
      ANI     L4033  ; 出料段  異常復歸
      OR      T3914  ; 出料手臂急停異常延遲
      ANB
      AND     L2871  ; Unload_ ROBOT_  CC-Link OK
      OUT     M4117  ; 出料手臂急停異常
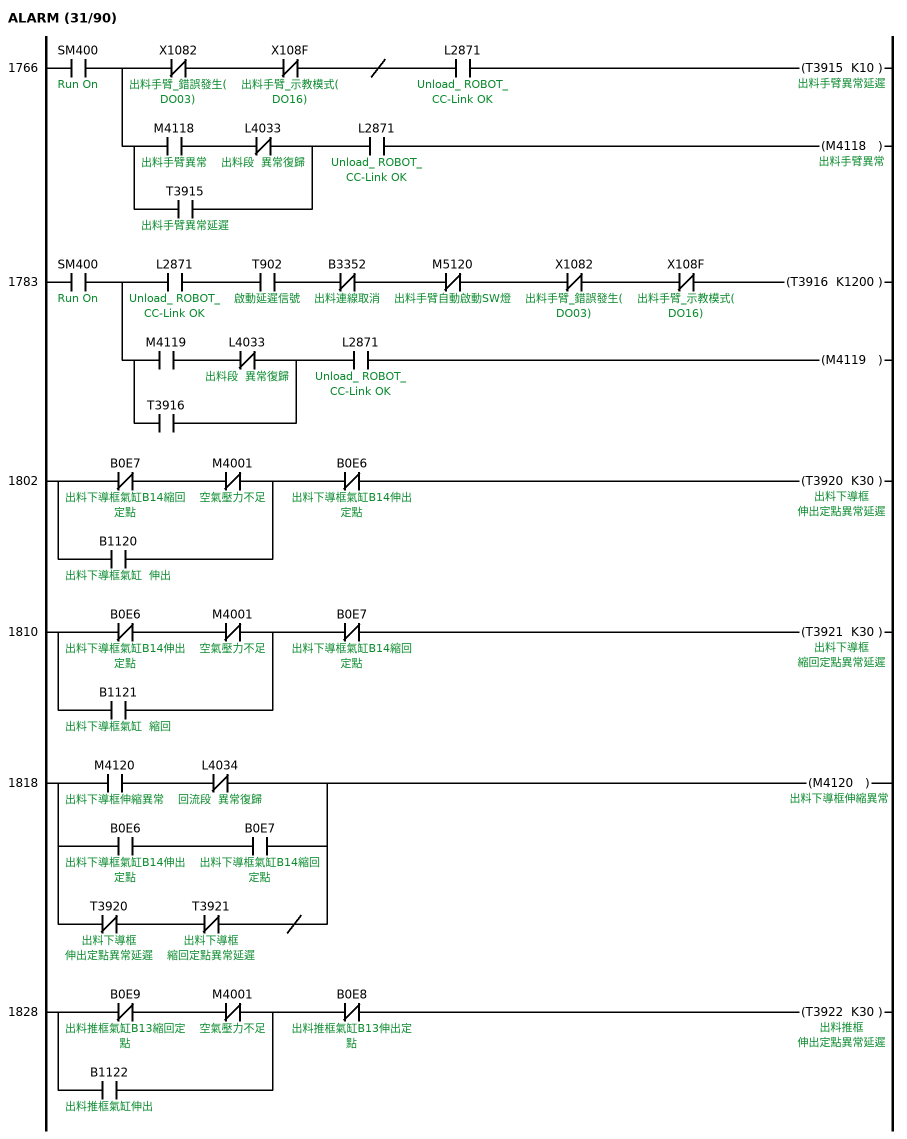
1766  LD      SM400  ; Run On
      MPS
      ANI     X1082  ; 出料手臂_錯誤發生(DO03)
      ANI     X108F  ; 出料手臂_示教模式(DO16)
      INV
      AND     L2871  ; Unload_ ROBOT_  CC-Link OK
      OUT     T3915 K10  ; 出料手臂異常延遲
      MPP
      LD      M4118  ; 出料手臂異常
      ANI     L4033  ; 出料段  異常復歸
      OR      T3915  ; 出料手臂異常延遲
      ANB
      AND     L2871  ; Unload_ ROBOT_  CC-Link OK
      OUT     M4118  ; 出料手臂異常
1783  LD      SM400  ; Run On
      MPS
      AND     L2871  ; Unload_ ROBOT_  CC-Link OK
      AND     T902  ; 啟動延遲信號
      ANI     B3352  ; 出料連線取消
      ANI     M5120  ; 出料手臂自動啟動SW燈
      ANI     X1082  ; 出料手臂_錯誤發生(DO03)
      ANI     X108F  ; 出料手臂_示教模式(DO16)
      OUT     T3916 K1200
      MPP
      LD      M4119
      ANI     L4033  ; 出料段  異常復歸
      OR      T3916
      ANB
      AND     L2871  ; Unload_ ROBOT_  CC-Link OK
      OUT     M4119
1802  LDI     B0E7  ; 出料下導框氣缸B14縮回定點
      ANI     M4001  ; 空氣壓力不足
      OR      B1120  ; 出料下導框氣缸  伸出
      ANI     B0E6  ; 出料下導框氣缸B14伸出定點
      OUT     T3920 K30  ; 出料下導框    伸出定點異常延遲
1810  LDI     B0E6  ; 出料下導框氣缸B14伸出定點
      ANI     M4001  ; 空氣壓力不足
      OR      B1121  ; 出料下導框氣缸  縮回
      ANI     B0E7  ; 出料下導框氣缸B14縮回定點
      OUT     T3921 K30  ; 出料下導框    縮回定點異常延遲
1818  LD      M4120  ; 出料下導框伸縮異常
      ANI     L4034  ; 回流段  異常復歸
      LD      B0E6  ; 出料下導框氣缸B14伸出定點
      AND     B0E7  ; 出料下導框氣缸B14縮回定點
      ORB
      LDI     T3920  ; 出料下導框    伸出定點異常延遲
      ANI     T3921  ; 出料下導框    縮回定點異常延遲
      INV
      ORB
      OUT     M4120  ; 出料下導框伸縮異常
1828  LDI     B0E9  ; 出料推框氣缸B13縮回定點
      ANI     M4001  ; 空氣壓力不足
      OR      B1122  ; 出料推框氣缸伸出
      ANI     B0E8  ; 出料推框氣缸B13伸出定點
      OUT     T3922 K30  ; 出料推框    伸出定點異常延遲
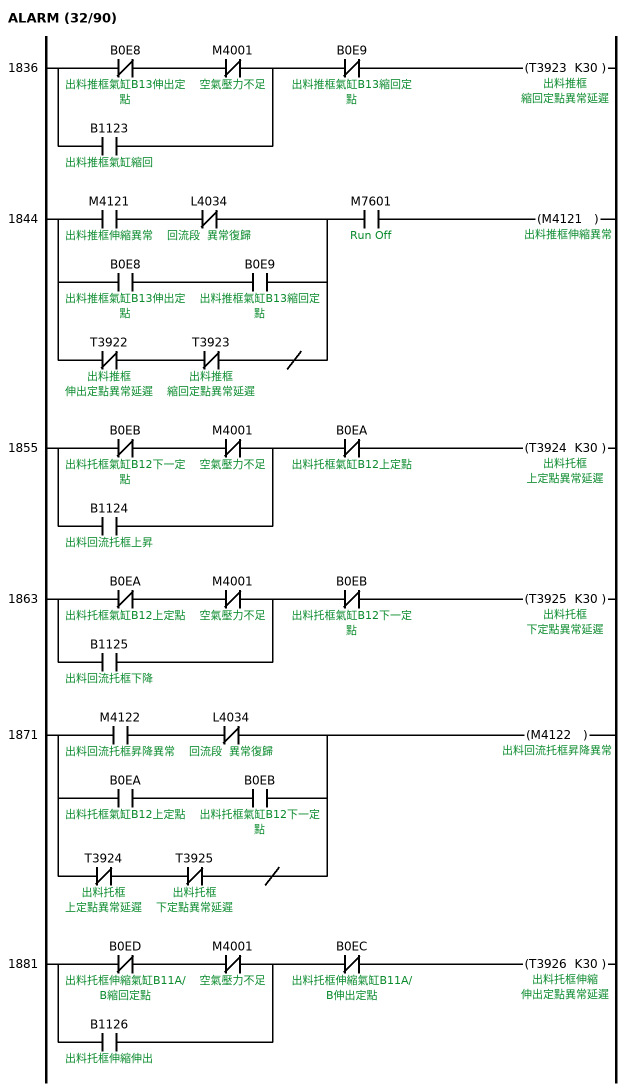
1836  LDI     B0E8  ; 出料推框氣缸B13伸出定點
      ANI     M4001  ; 空氣壓力不足
      OR      B1123  ; 出料推框氣缸縮回
      ANI     B0E9  ; 出料推框氣缸B13縮回定點
      OUT     T3923 K30  ; 出料推框    縮回定點異常延遲
1844  LD      M4121  ; 出料推框伸縮異常
      ANI     L4034  ; 回流段  異常復歸
      LD      B0E8  ; 出料推框氣缸B13伸出定點
      AND     B0E9  ; 出料推框氣缸B13縮回定點
      ORB
      LDI     T3922  ; 出料推框    伸出定點異常延遲
      ANI     T3923  ; 出料推框    縮回定點異常延遲
      INV
      ORB
      AND     M7601  ; Run Off
      OUT     M4121  ; 出料推框伸縮異常
1855  LDI     B0EB  ; 出料托框氣缸B12下一定點
      ANI     M4001  ; 空氣壓力不足
      OR      B1124  ; 出料回流托框上昇
      ANI     B0EA  ; 出料托框氣缸B12上定點
      OUT     T3924 K30  ; 出料托框    上定點異常延遲
1863  LDI     B0EA  ; 出料托框氣缸B12上定點
      ANI     M4001  ; 空氣壓力不足
      OR      B1125  ; 出料回流托框下降
      ANI     B0EB  ; 出料托框氣缸B12下一定點
      OUT     T3925 K30  ; 出料托框    下定點異常延遲
1871  LD      M4122  ; 出料回流托框昇降異常
      ANI     L4034  ; 回流段  異常復歸
      LD      B0EA  ; 出料托框氣缸B12上定點
      AND     B0EB  ; 出料托框氣缸B12下一定點
      ORB
      LDI     T3924  ; 出料托框    上定點異常延遲
      ANI     T3925  ; 出料托框    下定點異常延遲
      INV
      ORB
      OUT     M4122  ; 出料回流托框昇降異常
1881  LDI     B0ED  ; 出料托框伸縮氣缸B11A/B縮回定點
      ANI     M4001  ; 空氣壓力不足
      OR      B1126  ; 出料托框伸縮伸出
      ANI     B0EC  ; 出料托框伸縮氣缸B11A/B伸出定點
      OUT     T3926 K30  ; 出料托框伸縮    伸出定點異常延遲
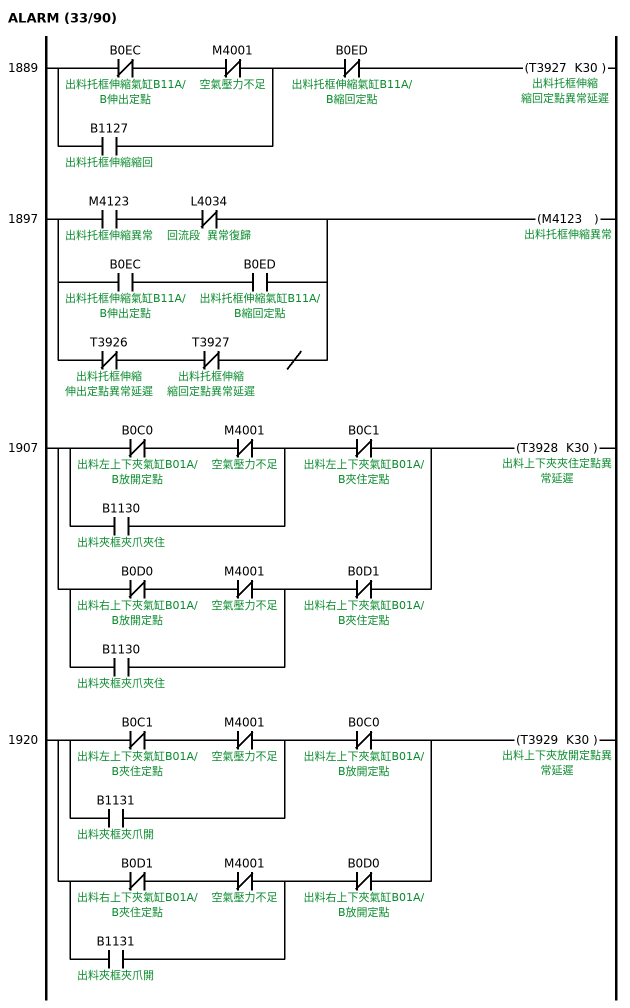
1889  LDI     B0EC  ; 出料托框伸縮氣缸B11A/B伸出定點
      ANI     M4001  ; 空氣壓力不足
      OR      B1127  ; 出料托框伸縮縮回
      ANI     B0ED  ; 出料托框伸縮氣缸B11A/B縮回定點
      OUT     T3927 K30  ; 出料托框伸縮    縮回定點異常延遲
1897  LD      M4123  ; 出料托框伸縮異常
      ANI     L4034  ; 回流段  異常復歸
      LD      B0EC  ; 出料托框伸縮氣缸B11A/B伸出定點
      AND     B0ED  ; 出料托框伸縮氣缸B11A/B縮回定點
      ORB
      LDI     T3926  ; 出料托框伸縮    伸出定點異常延遲
      ANI     T3927  ; 出料托框伸縮    縮回定點異常延遲
      INV
      ORB
      OUT     M4123  ; 出料托框伸縮異常
1907  LDI     B0C0  ; 出料左上下夾氣缸B01A/B放開定點
      ANI     M4001  ; 空氣壓力不足
      OR      B1130  ; 出料夾框夾爪夾住
      ANI     B0C1  ; 出料左上下夾氣缸B01A/B夾住定點
      LDI     B0D0  ; 出料右上下夾氣缸B01A/B放開定點
      ANI     M4001  ; 空氣壓力不足
      OR      B1130  ; 出料夾框夾爪夾住
      ANI     B0D1  ; 出料右上下夾氣缸B01A/B夾住定點
      ORB
      OUT     T3928 K30  ; 出料上下夾夾住定點異常延遲
1920  LDI     B0C1  ; 出料左上下夾氣缸B01A/B夾住定點
      ANI     M4001  ; 空氣壓力不足
      OR      B1131  ; 出料夾框夾爪開
      ANI     B0C0  ; 出料左上下夾氣缸B01A/B放開定點
      LDI     B0D1  ; 出料右上下夾氣缸B01A/B夾住定點
      ANI     M4001  ; 空氣壓力不足
      OR      B1131  ; 出料夾框夾爪開
      ANI     B0D0  ; 出料右上下夾氣缸B01A/B放開定點
      ORB
      OUT     T3929 K30  ; 出料上下夾放開定點異常延遲
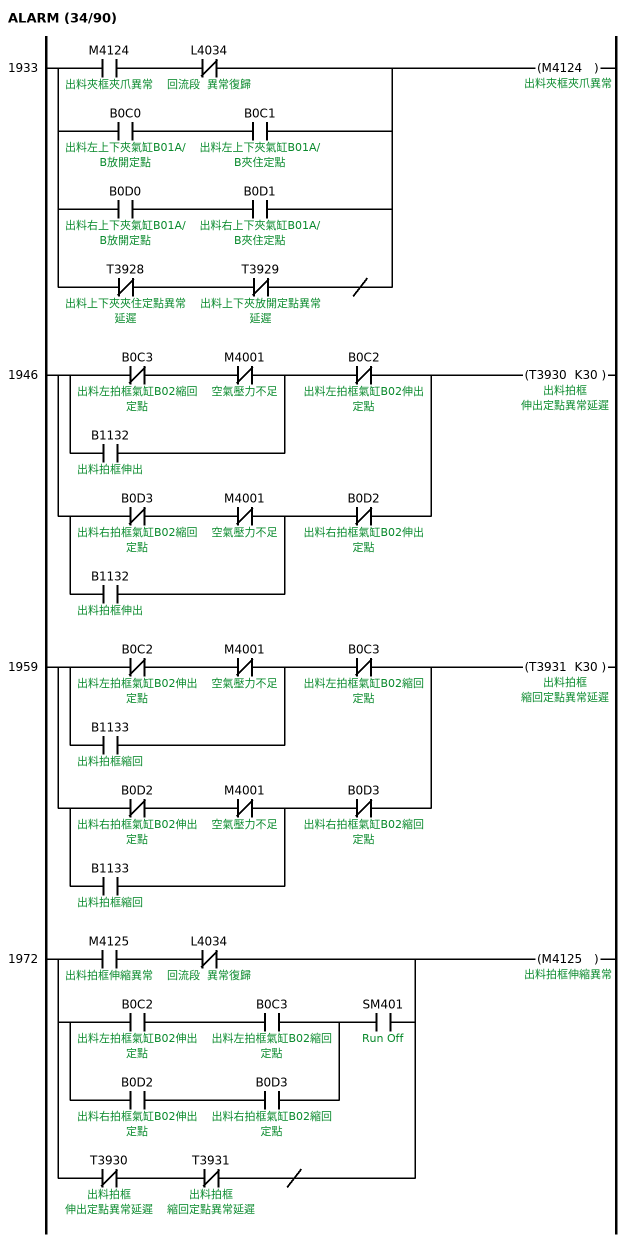
1933  LD      M4124  ; 出料夾框夾爪異常
      ANI     L4034  ; 回流段  異常復歸
      LD      B0C0  ; 出料左上下夾氣缸B01A/B放開定點
      AND     B0C1  ; 出料左上下夾氣缸B01A/B夾住定點
      ORB
      LD      B0D0  ; 出料右上下夾氣缸B01A/B放開定點
      AND     B0D1  ; 出料右上下夾氣缸B01A/B夾住定點
      ORB
      LDI     T3928  ; 出料上下夾夾住定點異常延遲
      ANI     T3929  ; 出料上下夾放開定點異常延遲
      INV
      ORB
      OUT     M4124  ; 出料夾框夾爪異常
1946  LDI     B0C3  ; 出料左拍框氣缸B02縮回定點
      ANI     M4001  ; 空氣壓力不足
      OR      B1132  ; 出料拍框伸出
      ANI     B0C2  ; 出料左拍框氣缸B02伸出定點
      LDI     B0D3  ; 出料右拍框氣缸B02縮回定點
      ANI     M4001  ; 空氣壓力不足
      OR      B1132  ; 出料拍框伸出
      ANI     B0D2  ; 出料右拍框氣缸B02伸出定點
      ORB
      OUT     T3930 K30  ; 出料拍框    伸出定點異常延遲
1959  LDI     B0C2  ; 出料左拍框氣缸B02伸出定點
      ANI     M4001  ; 空氣壓力不足
      OR      B1133  ; 出料拍框縮回
      ANI     B0C3  ; 出料左拍框氣缸B02縮回定點
      LDI     B0D2  ; 出料右拍框氣缸B02伸出定點
      ANI     M4001  ; 空氣壓力不足
      OR      B1133  ; 出料拍框縮回
      ANI     B0D3  ; 出料右拍框氣缸B02縮回定點
      ORB
      OUT     T3931 K30  ; 出料拍框    縮回定點異常延遲
1972  LD      M4125  ; 出料拍框伸縮異常
      ANI     L4034  ; 回流段  異常復歸
      LD      B0C2  ; 出料左拍框氣缸B02伸出定點
      AND     B0C3  ; 出料左拍框氣缸B02縮回定點
      LD      B0D2  ; 出料右拍框氣缸B02伸出定點
      AND     B0D3  ; 出料右拍框氣缸B02縮回定點
      ORB
      AND     SM401  ; Run Off
      ORB
      LDI     T3930  ; 出料拍框    伸出定點異常延遲
      ANI     T3931  ; 出料拍框    縮回定點異常延遲
      INV
      ORB
      OUT     M4125  ; 出料拍框伸縮異常
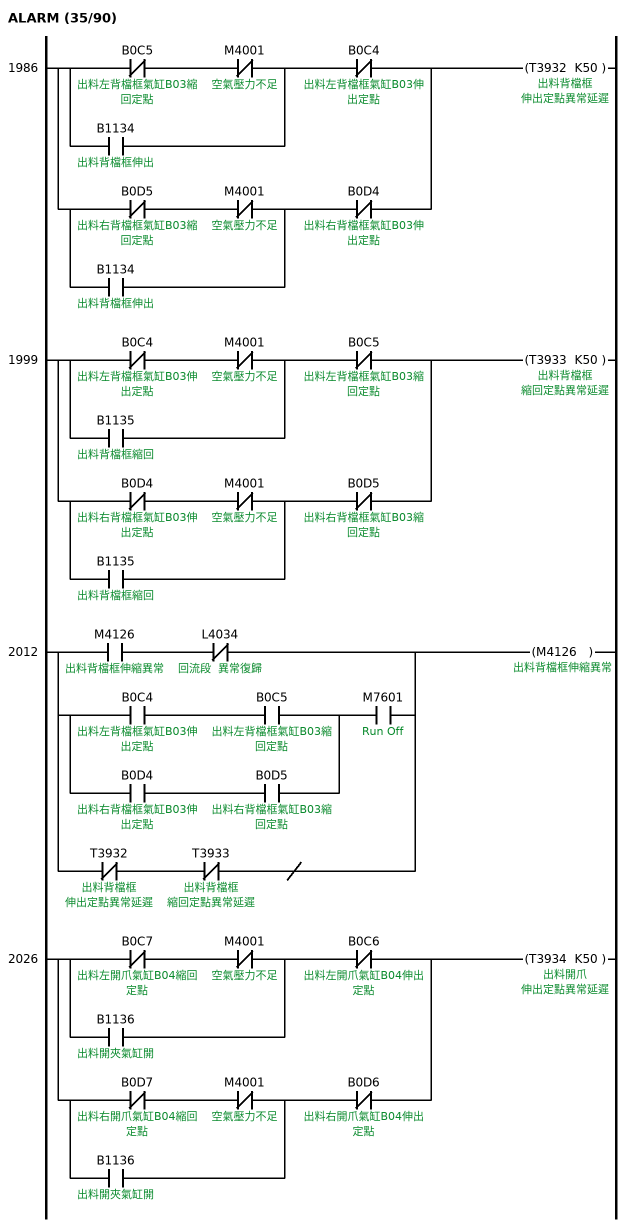
1986  LDI     B0C5  ; 出料左背檔框氣缸B03縮回定點
      ANI     M4001  ; 空氣壓力不足
      OR      B1134  ; 出料背檔框伸出
      ANI     B0C4  ; 出料左背檔框氣缸B03伸出定點
      LDI     B0D5  ; 出料右背檔框氣缸B03縮回定點
      ANI     M4001  ; 空氣壓力不足
      OR      B1134  ; 出料背檔框伸出
      ANI     B0D4  ; 出料右背檔框氣缸B03伸出定點
      ORB
      OUT     T3932 K50  ; 出料背檔框    伸出定點異常延遲
1999  LDI     B0C4  ; 出料左背檔框氣缸B03伸出定點
      ANI     M4001  ; 空氣壓力不足
      OR      B1135  ; 出料背檔框縮回
      ANI     B0C5  ; 出料左背檔框氣缸B03縮回定點
      LDI     B0D4  ; 出料右背檔框氣缸B03伸出定點
      ANI     M4001  ; 空氣壓力不足
      OR      B1135  ; 出料背檔框縮回
      ANI     B0D5  ; 出料右背檔框氣缸B03縮回定點
      ORB
      OUT     T3933 K50  ; 出料背檔框    縮回定點異常延遲
2012  LD      M4126  ; 出料背檔框伸縮異常
      ANI     L4034  ; 回流段  異常復歸
      LD      B0C4  ; 出料左背檔框氣缸B03伸出定點
      AND     B0C5  ; 出料左背檔框氣缸B03縮回定點
      LD      B0D4  ; 出料右背檔框氣缸B03伸出定點
      AND     B0D5  ; 出料右背檔框氣缸B03縮回定點
      ORB
      AND     M7601  ; Run Off
      ORB
      LDI     T3932  ; 出料背檔框    伸出定點異常延遲
      ANI     T3933  ; 出料背檔框    縮回定點異常延遲
      INV
      ORB
      OUT     M4126  ; 出料背檔框伸縮異常
2026  LDI     B0C7  ; 出料左開爪氣缸B04縮回定點
      ANI     M4001  ; 空氣壓力不足
      OR      B1136  ; 出料開夾氣缸開
      ANI     B0C6  ; 出料左開爪氣缸B04伸出定點
      LDI     B0D7  ; 出料右開爪氣缸B04縮回定點
      ANI     M4001  ; 空氣壓力不足
      OR      B1136  ; 出料開夾氣缸開
      ANI     B0D6  ; 出料右開爪氣缸B04伸出定點
      ORB
      OUT     T3934 K50  ; 出料開爪    伸出定點異常延遲
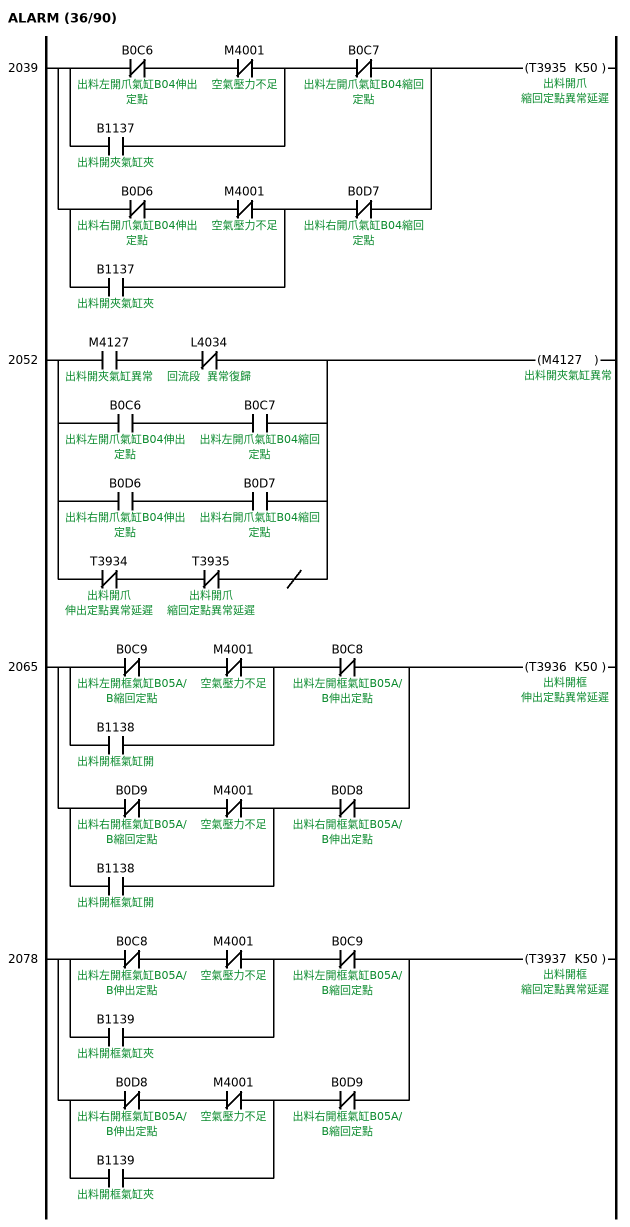
2039  LDI     B0C6  ; 出料左開爪氣缸B04伸出定點
      ANI     M4001  ; 空氣壓力不足
      OR      B1137  ; 出料開夾氣缸夾
      ANI     B0C7  ; 出料左開爪氣缸B04縮回定點
      LDI     B0D6  ; 出料右開爪氣缸B04伸出定點
      ANI     M4001  ; 空氣壓力不足
      OR      B1137  ; 出料開夾氣缸夾
      ANI     B0D7  ; 出料右開爪氣缸B04縮回定點
      ORB
      OUT     T3935 K50  ; 出料開爪    縮回定點異常延遲
2052  LD      M4127  ; 出料開夾氣缸異常
      ANI     L4034  ; 回流段  異常復歸
      LD      B0C6  ; 出料左開爪氣缸B04伸出定點
      AND     B0C7  ; 出料左開爪氣缸B04縮回定點
      ORB
      LD      B0D6  ; 出料右開爪氣缸B04伸出定點
      AND     B0D7  ; 出料右開爪氣缸B04縮回定點
      ORB
      LDI     T3934  ; 出料開爪    伸出定點異常延遲
      ANI     T3935  ; 出料開爪    縮回定點異常延遲
      INV
      ORB
      OUT     M4127  ; 出料開夾氣缸異常
2065  LDI     B0C9  ; 出料左開框氣缸B05A/B縮回定點
      ANI     M4001  ; 空氣壓力不足
      OR      B1138  ; 出料開框氣缸開
      ANI     B0C8  ; 出料左開框氣缸B05A/B伸出定點
      LDI     B0D9  ; 出料右開框氣缸B05A/B縮回定點
      ANI     M4001  ; 空氣壓力不足
      OR      B1138  ; 出料開框氣缸開
      ANI     B0D8  ; 出料右開框氣缸B05A/B伸出定點
      ORB
      OUT     T3936 K50  ; 出料開框    伸出定點異常延遲
2078  LDI     B0C8  ; 出料左開框氣缸B05A/B伸出定點
      ANI     M4001  ; 空氣壓力不足
      OR      B1139  ; 出料開框氣缸夾
      ANI     B0C9  ; 出料左開框氣缸B05A/B縮回定點
      LDI     B0D8  ; 出料右開框氣缸B05A/B伸出定點
      ANI     M4001  ; 空氣壓力不足
      OR      B1139  ; 出料開框氣缸夾
      ANI     B0D9  ; 出料右開框氣缸B05A/B縮回定點
      ORB
      OUT     T3937 K50  ; 出料開框    縮回定點異常延遲
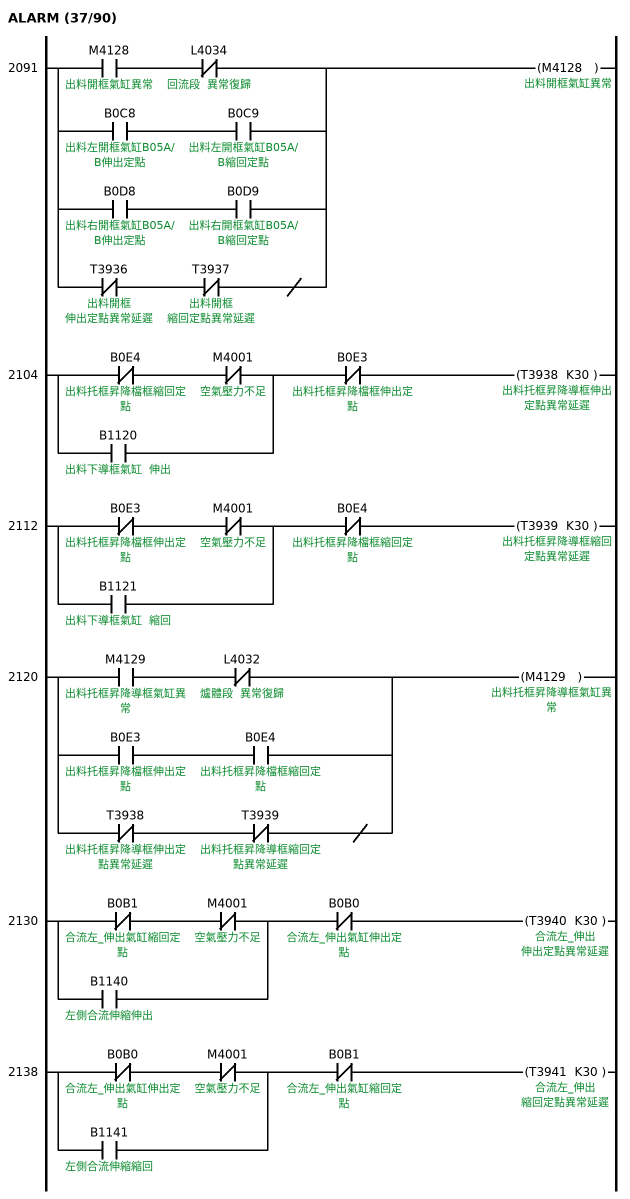
2091  LD      M4128  ; 出料開框氣缸異常
      ANI     L4034  ; 回流段  異常復歸
      LD      B0C8  ; 出料左開框氣缸B05A/B伸出定點
      AND     B0C9  ; 出料左開框氣缸B05A/B縮回定點
      ORB
      LD      B0D8  ; 出料右開框氣缸B05A/B伸出定點
      AND     B0D9  ; 出料右開框氣缸B05A/B縮回定點
      ORB
      LDI     T3936  ; 出料開框    伸出定點異常延遲
      ANI     T3937  ; 出料開框    縮回定點異常延遲
      INV
      ORB
      OUT     M4128  ; 出料開框氣缸異常
2104  LDI     B0E4  ; 出料托框昇降檔框縮回定點
      ANI     M4001  ; 空氣壓力不足
      OR      B1120  ; 出料下導框氣缸  伸出
      ANI     B0E3  ; 出料托框昇降檔框伸出定點
      OUT     T3938 K30  ; 出料托框昇降導框伸出定點異常延遲
2112  LDI     B0E3  ; 出料托框昇降檔框伸出定點
      ANI     M4001  ; 空氣壓力不足
      OR      B1121  ; 出料下導框氣缸  縮回
      ANI     B0E4  ; 出料托框昇降檔框縮回定點
      OUT     T3939 K30  ; 出料托框昇降導框縮回定點異常延遲
2120  LD      M4129  ; 出料托框昇降導框氣缸異常
      ANI     L4032  ; 爐體段  異常復歸
      LD      B0E3  ; 出料托框昇降檔框伸出定點
      AND     B0E4  ; 出料托框昇降檔框縮回定點
      ORB
      LDI     T3938  ; 出料托框昇降導框伸出定點異常延遲
      ANI     T3939  ; 出料托框昇降導框縮回定點異常延遲
      INV
      ORB
      OUT     M4129  ; 出料托框昇降導框氣缸異常
2130  LDI     B0B1  ; 合流左_伸出氣缸縮回定點
      ANI     M4001  ; 空氣壓力不足
      OR      B1140  ; 左側合流伸縮伸出
      ANI     B0B0  ; 合流左_伸出氣缸伸出定點
      OUT     T3940 K30  ; 合流左_伸出    伸出定點異常延遲
2138  LDI     B0B0  ; 合流左_伸出氣缸伸出定點
      ANI     M4001  ; 空氣壓力不足
      OR      B1141  ; 左側合流伸縮縮回
      ANI     B0B1  ; 合流左_伸出氣缸縮回定點
      OUT     T3941 K30  ; 合流左_伸出    縮回定點異常延遲
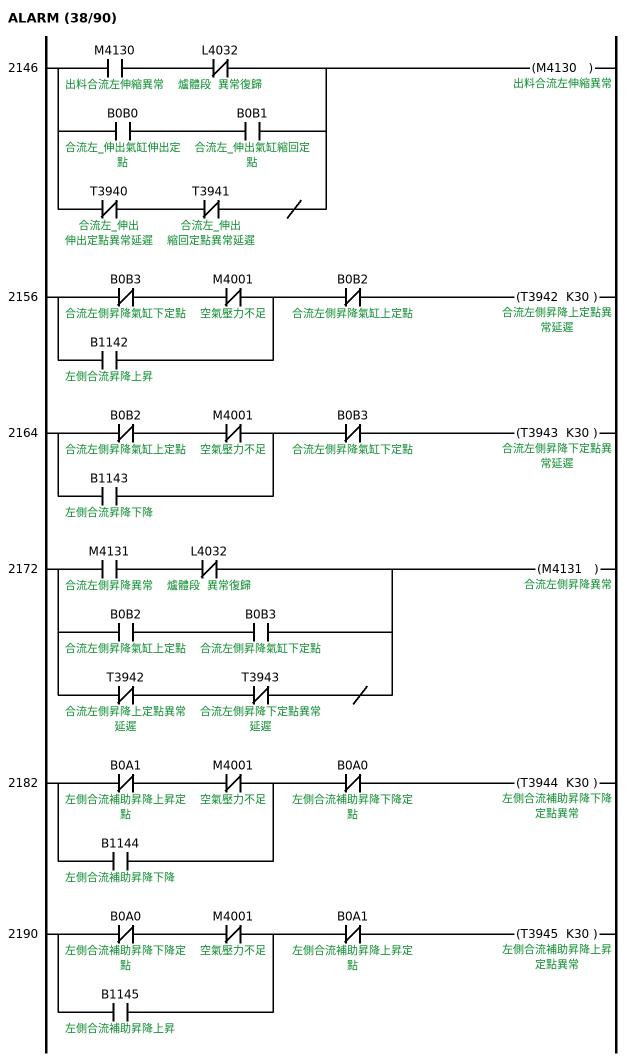
2146  LD      M4130  ; 出料合流左伸縮異常
      ANI     L4032  ; 爐體段  異常復歸
      LD      B0B0  ; 合流左_伸出氣缸伸出定點
      AND     B0B1  ; 合流左_伸出氣缸縮回定點
      ORB
      LDI     T3940  ; 合流左_伸出    伸出定點異常延遲
      ANI     T3941  ; 合流左_伸出    縮回定點異常延遲
      INV
      ORB
      OUT     M4130  ; 出料合流左伸縮異常
2156  LDI     B0B3  ; 合流左側昇降氣缸下定點
      ANI     M4001  ; 空氣壓力不足
      OR      B1142  ; 左側合流昇降上昇
      ANI     B0B2  ; 合流左側昇降氣缸上定點
      OUT     T3942 K30  ; 合流左側昇降上定點異常延遲
2164  LDI     B0B2  ; 合流左側昇降氣缸上定點
      ANI     M4001  ; 空氣壓力不足
      OR      B1143  ; 左側合流昇降下降
      ANI     B0B3  ; 合流左側昇降氣缸下定點
      OUT     T3943 K30  ; 合流左側昇降下定點異常延遲
2172  LD      M4131  ; 合流左側昇降異常
      ANI     L4032  ; 爐體段  異常復歸
      LD      B0B2  ; 合流左側昇降氣缸上定點
      AND     B0B3  ; 合流左側昇降氣缸下定點
      ORB
      LDI     T3942  ; 合流左側昇降上定點異常延遲
      ANI     T3943  ; 合流左側昇降下定點異常延遲
      INV
      ORB
      OUT     M4131  ; 合流左側昇降異常
2182  LDI     B0A1  ; 左側合流補助昇降上昇定點
      ANI     M4001  ; 空氣壓力不足
      OR      B1144  ; 左側合流補助昇降下降
      ANI     B0A0  ; 左側合流補助昇降下降定點
      OUT     T3944 K30  ; 左側合流補助昇降下降定點異常
2190  LDI     B0A0  ; 左側合流補助昇降下降定點
      ANI     M4001  ; 空氣壓力不足
      OR      B1145  ; 左側合流補助昇降上昇
      ANI     B0A1  ; 左側合流補助昇降上昇定點
      OUT     T3945 K30  ; 左側合流補助昇降上昇定點異常
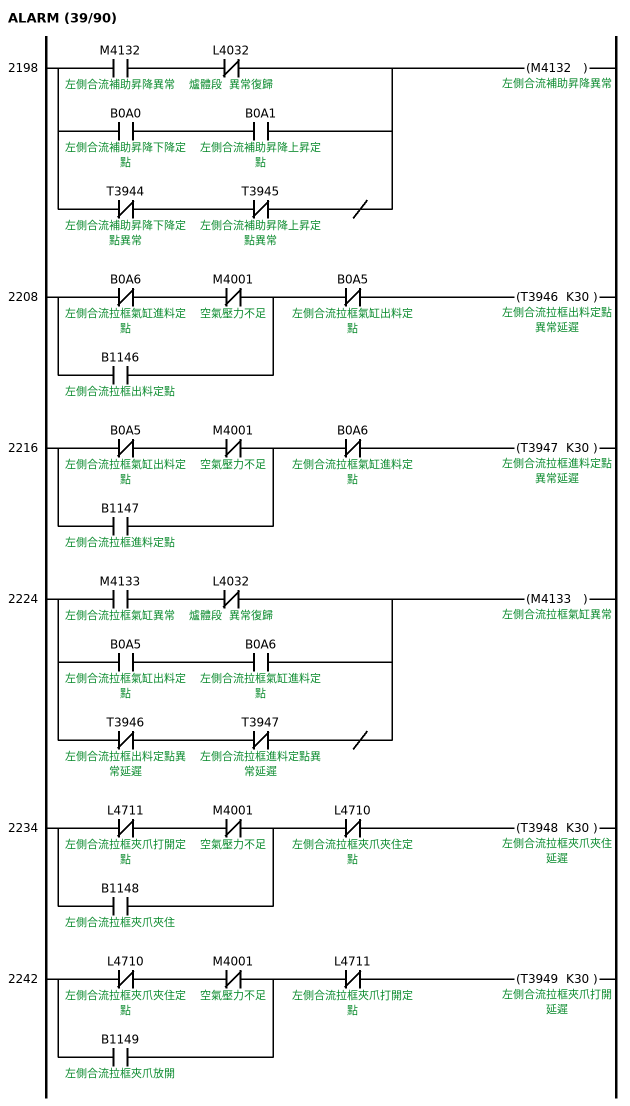
2198  LD      M4132  ; 左側合流補助昇降異常
      ANI     L4032  ; 爐體段  異常復歸
      LD      B0A0  ; 左側合流補助昇降下降定點
      AND     B0A1  ; 左側合流補助昇降上昇定點
      ORB
      LDI     T3944  ; 左側合流補助昇降下降定點異常
      ANI     T3945  ; 左側合流補助昇降上昇定點異常
      INV
      ORB
      OUT     M4132  ; 左側合流補助昇降異常
2208  LDI     B0A6  ; 左側合流拉框氣缸進料定點
      ANI     M4001  ; 空氣壓力不足
      OR      B1146  ; 左側合流拉框出料定點
      ANI     B0A5  ; 左側合流拉框氣缸出料定點
      OUT     T3946 K30  ; 左側合流拉框出料定點異常延遲
2216  LDI     B0A5  ; 左側合流拉框氣缸出料定點
      ANI     M4001  ; 空氣壓力不足
      OR      B1147  ; 左側合流拉框進料定點
      ANI     B0A6  ; 左側合流拉框氣缸進料定點
      OUT     T3947 K30  ; 左側合流拉框進料定點異常延遲
2224  LD      M4133  ; 左側合流拉框氣缸異常
      ANI     L4032  ; 爐體段  異常復歸
      LD      B0A5  ; 左側合流拉框氣缸出料定點
      AND     B0A6  ; 左側合流拉框氣缸進料定點
      ORB
      LDI     T3946  ; 左側合流拉框出料定點異常延遲
      ANI     T3947  ; 左側合流拉框進料定點異常延遲
      INV
      ORB
      OUT     M4133  ; 左側合流拉框氣缸異常
2234  LDI     L4711  ; 左側合流拉框夾爪打開定點
      ANI     M4001  ; 空氣壓力不足
      OR      B1148  ; 左側合流拉框夾爪夾住
      ANI     L4710  ; 左側合流拉框夾爪夾住定點
      OUT     T3948 K30  ; 左側合流拉框夾爪夾住延遲
2242  LDI     L4710  ; 左側合流拉框夾爪夾住定點
      ANI     M4001  ; 空氣壓力不足
      OR      B1149  ; 左側合流拉框夾爪放開
      ANI     L4711  ; 左側合流拉框夾爪打開定點
      OUT     T3949 K30  ; 左側合流拉框夾爪打開延遲
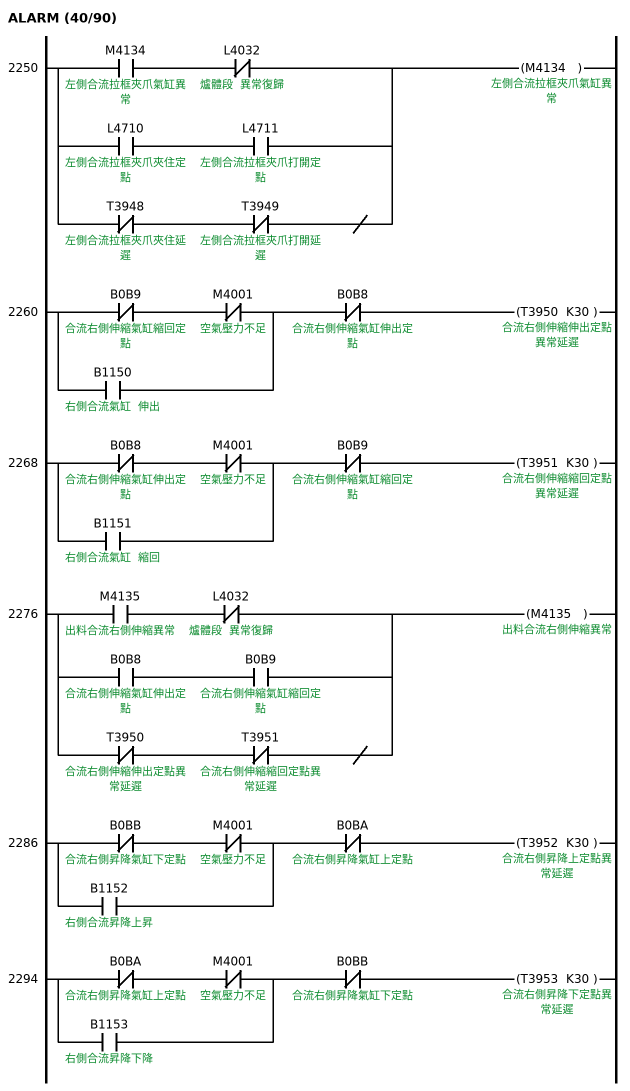
2250  LD      M4134  ; 左側合流拉框夾爪氣缸異常
      ANI     L4032  ; 爐體段  異常復歸
      LD      L4710  ; 左側合流拉框夾爪夾住定點
      AND     L4711  ; 左側合流拉框夾爪打開定點
      ORB
      LDI     T3948  ; 左側合流拉框夾爪夾住延遲
      ANI     T3949  ; 左側合流拉框夾爪打開延遲
      INV
      ORB
      OUT     M4134  ; 左側合流拉框夾爪氣缸異常
2260  LDI     B0B9  ; 合流右側伸縮氣缸縮回定點
      ANI     M4001  ; 空氣壓力不足
      OR      B1150  ; 右側合流氣缸  伸出
      ANI     B0B8  ; 合流右側伸縮氣缸伸出定點
      OUT     T3950 K30  ; 合流右側伸縮伸出定點異常延遲
2268  LDI     B0B8  ; 合流右側伸縮氣缸伸出定點
      ANI     M4001  ; 空氣壓力不足
      OR      B1151  ; 右側合流氣缸  縮回
      ANI     B0B9  ; 合流右側伸縮氣缸縮回定點
      OUT     T3951 K30  ; 合流右側伸縮縮回定點異常延遲
2276  LD      M4135  ; 出料合流右側伸縮異常
      ANI     L4032  ; 爐體段  異常復歸
      LD      B0B8  ; 合流右側伸縮氣缸伸出定點
      AND     B0B9  ; 合流右側伸縮氣缸縮回定點
      ORB
      LDI     T3950  ; 合流右側伸縮伸出定點異常延遲
      ANI     T3951  ; 合流右側伸縮縮回定點異常延遲
      INV
      ORB
      OUT     M4135  ; 出料合流右側伸縮異常
2286  LDI     B0BB  ; 合流右側昇降氣缸下定點
      ANI     M4001  ; 空氣壓力不足
      OR      B1152  ; 右側合流昇降上昇
      ANI     B0BA  ; 合流右側昇降氣缸上定點
      OUT     T3952 K30  ; 合流右側昇降上定點異常延遲
2294  LDI     B0BA  ; 合流右側昇降氣缸上定點
      ANI     M4001  ; 空氣壓力不足
      OR      B1153  ; 右側合流昇降下降
      ANI     B0BB  ; 合流右側昇降氣缸下定點
      OUT     T3953 K30  ; 合流右側昇降下定點異常延遲
